   1:  PR[GP1:91,1] = PR[GP1:90,1] + -41.050;
   1:  PR[GP1:91,2] = PR[GP1:90,2] + 5.137;
   1:L PR[91] R[100]mm/sec CNT100;
   1:  PR[GP1:91,1] = PR[GP1:90,1] + -41.412;
   1:  PR[GP1:91,2] = PR[GP1:90,2] + 3.695;
   1:L PR[91] R[100]mm/sec CNT100;
   1:  PR[GP1:91,1] = PR[GP1:90,1] + -41.545;
   1:  PR[GP1:91,2] = PR[GP1:90,2] + 2.074;
   1:L PR[91] R[100]mm/sec CNT100;
   1:  PR[GP1:91,1] = PR[GP1:90,1] + -41.859;
   1:  PR[GP1:91,2] = PR[GP1:90,2] + -0.346;
   1:L PR[91] R[100]mm/sec CNT100;
   1:  PR[GP1:91,1] = PR[GP1:90,1] + -41.730;
   1:  PR[GP1:91,2] = PR[GP1:90,2] + -1.916;
   1:L PR[91] R[100]mm/sec CNT100;
   1:  PR[GP1:91,1] = PR[GP1:90,1] + -41.420;
   1:  PR[GP1:91,2] = PR[GP1:90,2] + -4.285;
   1:L PR[91] R[100]mm/sec CNT100;
   1:  PR[GP1:91,1] = PR[GP1:90,1] + -41.054;
   1:  PR[GP1:91,2] = PR[GP1:90,2] + -5.749;
   1:L PR[91] R[100]mm/sec CNT100;
   1:  PR[GP1:91,1] = PR[GP1:90,1] + -40.415;
   1:  PR[GP1:91,2] = PR[GP1:90,2] + -7.221;
   1:L PR[91] R[100]mm/sec CNT100;
   1:  PR[GP1:91,1] = PR[GP1:90,1] + -39.483;
   1:  PR[GP1:91,2] = PR[GP1:90,2] + -9.478;
   1:L PR[91] R[100]mm/sec CNT100;
   1:  PR[GP1:91,1] = PR[GP1:90,1] + -38.675;
   1:  PR[GP1:91,2] = PR[GP1:90,2] + -10.730;
   1:L PR[91] R[100]mm/sec CNT100;
   1:  PR[GP1:91,1] = PR[GP1:90,1] + -37.137;
   1:  PR[GP1:91,2] = PR[GP1:90,2] + -12.747;
   1:L PR[91] R[100]mm/sec CNT100;
   1:  PR[GP1:91,1] = PR[GP1:90,1] + -36.167;
   1:  PR[GP1:91,2] = PR[GP1:90,2] + -13.817;
   1:L PR[91] R[100]mm/sec CNT100;
   1:  PR[GP1:91,1] = PR[GP1:90,1] + -34.995;
   1:  PR[GP1:91,2] = PR[GP1:90,2] + -14.746;
   1:L PR[91] R[100]mm/sec CNT100;
   1:  PR[GP1:91,1] = PR[GP1:90,1] + -32.930;
   1:  PR[GP1:91,2] = PR[GP1:90,2] + -16.344;
   1:L PR[91] R[100]mm/sec CNT100;
   1:  PR[GP1:91,1] = PR[GP1:90,1] + -31.743;
   1:  PR[GP1:91,2] = PR[GP1:90,2] + -17.003;
   1:L PR[91] R[100]mm/sec CNT100;
   1:  PR[GP1:91,1] = PR[GP1:90,1] + -29.159;
   1:  PR[GP1:91,2] = PR[GP1:90,2] + -18.091;
   1:L PR[91] R[100]mm/sec CNT100;
   1:  PR[GP1:91,1] = PR[GP1:90,1] + -27.947;
   1:  PR[GP1:91,2] = PR[GP1:90,2] + -18.524;
   1:L PR[91] R[100]mm/sec CNT100;
   1:  PR[GP1:91,1] = PR[GP1:90,1] + -26.670;
   1:  PR[GP1:91,2] = PR[GP1:90,2] + -18.756;
   1:L PR[91] R[100]mm/sec CNT100;
   1:  PR[GP1:91,1] = PR[GP1:90,1] + -23.763;
   1:  PR[GP1:91,2] = PR[GP1:90,2] + -19.163;
   1:L PR[91] R[100]mm/sec CNT100;
   1:  PR[GP1:91,1] = PR[GP1:90,1] + -22.646;
   1:  PR[GP1:91,2] = PR[GP1:90,2] + -19.180;
   1:L PR[91] R[100]mm/sec CNT100;
   1:  PR[GP1:91,1] = PR[GP1:90,1] + -21.433;
   1:  PR[GP1:91,2] = PR[GP1:90,2] + -18.999;
   1:L PR[91] R[100]mm/sec CNT100;
   1:  PR[GP1:91,1] = PR[GP1:90,1] + -18.373;
   1:  PR[GP1:91,2] = PR[GP1:90,2] + -18.633;
   1:L PR[91] R[100]mm/sec CNT100;
   1:  PR[GP1:91,1] = PR[GP1:90,1] + -17.424;
   1:  PR[GP1:91,2] = PR[GP1:90,2] + -18.327;
   1:L PR[91] R[100]mm/sec CNT100;
   1:  PR[GP1:91,1] = PR[GP1:90,1] + -14.274;
   1:  PR[GP1:91,2] = PR[GP1:90,2] + -17.068;
   1:L PR[91] R[100]mm/sec CNT100;
   1:  PR[GP1:91,1] = PR[GP1:90,1] + -13.518;
   1:  PR[GP1:91,2] = PR[GP1:90,2] + -16.679;
   1:L PR[91] R[100]mm/sec CNT100;
   1:  PR[GP1:91,1] = PR[GP1:90,1] + -9.919;
   1:  PR[GP1:91,2] = PR[GP1:90,2] + -14.005;
   1:L PR[91] R[100]mm/sec CNT100;
   1:  PR[GP1:91,1] = PR[GP1:90,1] + -9.431;
   1:  PR[GP1:91,2] = PR[GP1:90,2] + -13.499;
   1:L PR[91] R[100]mm/sec CNT100;
   1:  PR[GP1:91,1] = PR[GP1:90,1] + -7.028;
   1:  PR[GP1:91,2] = PR[GP1:90,2] + -10.470;
   1:L PR[91] R[100]mm/sec CNT100;
   1:  PR[GP1:91,1] = PR[GP1:90,1] + -6.688;
   1:  PR[GP1:91,2] = PR[GP1:90,2] + -9.977;
   1:L PR[91] R[100]mm/sec CNT100;
   1:  PR[GP1:91,1] = PR[GP1:90,1] + -6.421;
   1:  PR[GP1:91,2] = PR[GP1:90,2] + -9.412;
   1:L PR[91] R[100]mm/sec CNT100;
   1:  PR[GP1:91,1] = PR[GP1:90,1] + -4.821;
   1:  PR[GP1:91,2] = PR[GP1:90,2] + -5.735;
   1:L PR[91] R[100]mm/sec CNT100;
   1:  PR[GP1:91,1] = PR[GP1:90,1] + -4.521;
   1:  PR[GP1:91,2] = PR[GP1:90,2] + -4.703;
   1:L PR[91] R[100]mm/sec CNT100;
   1:  PR[GP1:91,1] = PR[GP1:90,1] + -4.126;
   1:  PR[GP1:91,2] = PR[GP1:90,2] + -4.264;
   1:L PR[91] R[100]mm/sec CNT100;
   1:  PR[GP1:91,1] = PR[GP1:90,1] + -3.629;
   1:  PR[GP1:91,2] = PR[GP1:90,2] + -3.586;
   1:L PR[91] R[100]mm/sec CNT100;
   1:  PR[GP1:91,1] = PR[GP1:90,1] + -2.653;
   1:  PR[GP1:91,2] = PR[GP1:90,2] + -2.949;
   1:L PR[91] R[100]mm/sec CNT100;
   1:  PR[GP1:91,1] = PR[GP1:90,1] + -1.650;
   1:  PR[GP1:91,2] = PR[GP1:90,2] + -2.748;
   1:L PR[91] R[100]mm/sec CNT100;
   1:  PR[GP1:91,1] = PR[GP1:90,1] + 1.800;
   1:L PR[91] R[100]mm/sec CNT100;
   1:  PR[GP1:91,1] = PR[GP1:90,1] + 2.807;
   1:  PR[GP1:91,2] = PR[GP1:90,2] + -2.948;
   1:L PR[91] R[100]mm/sec CNT100;
   1:  PR[GP1:91,1] = PR[GP1:90,1] + 3.784;
   1:  PR[GP1:91,2] = PR[GP1:90,2] + -3.585;
   1:L PR[91] R[100]mm/sec CNT100;
   1:  PR[GP1:91,1] = PR[GP1:90,1] + 4.289;
   1:  PR[GP1:91,2] = PR[GP1:90,2] + -4.274;
   1:L PR[91] R[100]mm/sec CNT100;
   1:  PR[GP1:91,1] = PR[GP1:90,1] + 4.700;
   1:  PR[GP1:91,2] = PR[GP1:90,2] + -4.748;
   1:L PR[91] R[100]mm/sec CNT100;
   1:  PR[GP1:91,1] = PR[GP1:90,1] + 4.937;
   1:  PR[GP1:91,2] = PR[GP1:90,2] + -5.561;
   1:L PR[91] R[100]mm/sec CNT100;
   1:  PR[GP1:91,1] = PR[GP1:90,1] + 5.121;
   1:  PR[GP1:91,2] = PR[GP1:90,2] + -5.951;
   1:L PR[91] R[100]mm/sec CNT100;
   1:  PR[GP1:91,1] = PR[GP1:90,1] + 6.858;
   1:  PR[GP1:91,2] = PR[GP1:90,2] + -9.995;
   1:L PR[91] R[100]mm/sec CNT100;
   1:  PR[GP1:91,1] = PR[GP1:90,1] + 7.184;
   1:  PR[GP1:91,2] = PR[GP1:90,2] + -10.467;
   1:L PR[91] R[100]mm/sec CNT100;
   1:  PR[GP1:91,1] = PR[GP1:90,1] + 9.586;
   1:  PR[GP1:91,2] = PR[GP1:90,2] + -13.499;
   1:L PR[91] R[100]mm/sec CNT100;
   1:  PR[GP1:91,1] = PR[GP1:90,1] + 10.074;
   1:  PR[GP1:91,2] = PR[GP1:90,2] + -14.004;
   1:L PR[91] R[100]mm/sec CNT100;
   1:  PR[GP1:91,1] = PR[GP1:90,1] + 13.674;
   1:  PR[GP1:91,2] = PR[GP1:90,2] + -16.678;
   1:L PR[91] R[100]mm/sec CNT100;
   1:  PR[GP1:91,1] = PR[GP1:90,1] + 14.429;
   1:  PR[GP1:91,2] = PR[GP1:90,2] + -17.068;
   1:L PR[91] R[100]mm/sec CNT100;
   1:  PR[GP1:91,1] = PR[GP1:90,1] + 17.579;
   1:  PR[GP1:91,2] = PR[GP1:90,2] + -18.327;
   1:L PR[91] R[100]mm/sec CNT100;
   1:  PR[GP1:91,1] = PR[GP1:90,1] + 18.548;
   1:  PR[GP1:91,2] = PR[GP1:90,2] + -18.639;
   1:L PR[91] R[100]mm/sec CNT100;
   1:  PR[GP1:91,1] = PR[GP1:90,1] + 19.584;
   1:  PR[GP1:91,2] = PR[GP1:90,2] + -18.793;
   1:L PR[91] R[100]mm/sec CNT100;
   1:  PR[GP1:91,1] = PR[GP1:90,1] + 22.782;
   1:  PR[GP1:91,2] = PR[GP1:90,2] + -19.181;
   1:L PR[91] R[100]mm/sec CNT100;
   1:  PR[GP1:91,1] = PR[GP1:90,1] + 23.889;
   1:  PR[GP1:91,2] = PR[GP1:90,2] + -19.163;
   1:L PR[91] R[100]mm/sec CNT100;
   1:  PR[GP1:91,1] = PR[GP1:90,1] + 25.103;
   1:  PR[GP1:91,2] = PR[GP1:90,2] + -18.943;
   1:L PR[91] R[100]mm/sec CNT100;
   1:  PR[GP1:91,1] = PR[GP1:90,1] + 28.130;
   1:  PR[GP1:91,2] = PR[GP1:90,2] + -18.515;
   1:L PR[91] R[100]mm/sec CNT100;
   1:  PR[GP1:91,1] = PR[GP1:90,1] + 29.315;
   1:  PR[GP1:91,2] = PR[GP1:90,2] + -18.091;
   1:L PR[91] R[100]mm/sec CNT100;
   1:  PR[GP1:91,1] = PR[GP1:90,1] + 31.900;
   1:  PR[GP1:91,2] = PR[GP1:90,2] + -17.004;
   1:L PR[91] R[100]mm/sec CNT100;
   1:  PR[GP1:91,1] = PR[GP1:90,1] + 33.079;
   1:  PR[GP1:91,2] = PR[GP1:90,2] + -16.349;
   1:L PR[91] R[100]mm/sec CNT100;
   1:  PR[GP1:91,1] = PR[GP1:90,1] + 34.204;
   1:  PR[GP1:91,2] = PR[GP1:90,2] + -15.457;
   1:L PR[91] R[100]mm/sec CNT100;
   1:  PR[GP1:91,1] = PR[GP1:90,1] + 36.329;
   1:  PR[GP1:91,2] = PR[GP1:90,2] + -13.811;
   1:L PR[91] R[100]mm/sec CNT100;
   1:  PR[GP1:91,1] = PR[GP1:90,1] + 37.293;
   1:  PR[GP1:91,2] = PR[GP1:90,2] + -12.748;
   1:L PR[91] R[100]mm/sec CNT100;
   1:  PR[GP1:91,1] = PR[GP1:90,1] + 38.832;
   1:  PR[GP1:91,2] = PR[GP1:90,2] + -10.730;
   1:L PR[91] R[100]mm/sec CNT100;
   1:  PR[GP1:91,1] = PR[GP1:90,1] + 39.647;
   1:  PR[GP1:91,2] = PR[GP1:90,2] + -9.467;
   1:L PR[91] R[100]mm/sec CNT100;
   1:  PR[GP1:91,1] = PR[GP1:90,1] + 40.262;
   1:  PR[GP1:91,2] = PR[GP1:90,2] + -8.047;
   1:L PR[91] R[100]mm/sec CNT100;
   1:  PR[GP1:91,1] = PR[GP1:90,1] + 41.207;
   1:  PR[GP1:91,2] = PR[GP1:90,2] + -5.762;
   1:L PR[91] R[100]mm/sec CNT100;
   1:  PR[GP1:91,1] = PR[GP1:90,1] + 41.569;
   1:  PR[GP1:91,2] = PR[GP1:90,2] + -4.320;
   1:L PR[91] R[100]mm/sec CNT100;
   1:  PR[GP1:91,1] = PR[GP1:90,1] + 41.702;
   1:  PR[GP1:91,2] = PR[GP1:90,2] + -2.699;
   1:L PR[91] R[100]mm/sec CNT100;
   1:  PR[GP1:91,1] = PR[GP1:90,1] + 42.016;
   1:  PR[GP1:91,2] = PR[GP1:90,2] + -0.278;
   1:L PR[91] R[100]mm/sec CNT100;
   1:  PR[GP1:91,1] = PR[GP1:90,1] + 41.887;
   1:  PR[GP1:91,2] = PR[GP1:90,2] + 1.292;
   1:L PR[91] R[100]mm/sec CNT100;
   1:  PR[GP1:91,1] = PR[GP1:90,1] + 41.577;
   1:  PR[GP1:91,2] = PR[GP1:90,2] + 3.663;
   1:L PR[91] R[100]mm/sec CNT100;
   1:  PR[GP1:91,1] = PR[GP1:90,1] + 41.210;
   1:  PR[GP1:91,2] = PR[GP1:90,2] + 5.127;
   1:L PR[91] R[100]mm/sec CNT100;
   1:  PR[GP1:91,1] = PR[GP1:90,1] + 40.572;
   1:  PR[GP1:91,2] = PR[GP1:90,2] + 6.599;
   1:L PR[91] R[100]mm/sec CNT100;
   1:  PR[GP1:91,1] = PR[GP1:90,1] + 39.639;
   1:  PR[GP1:91,2] = PR[GP1:90,2] + 8.854;
   1:L PR[91] R[100]mm/sec CNT100;
   1:  PR[GP1:91,1] = PR[GP1:90,1] + 38.831;
   1:  PR[GP1:91,2] = PR[GP1:90,2] + 10.107;
   1:L PR[91] R[100]mm/sec CNT100;
   1:  PR[GP1:91,1] = PR[GP1:90,1] + 37.292;
   1:  PR[GP1:91,2] = PR[GP1:90,2] + 12.125;
   1:L PR[91] R[100]mm/sec CNT100;
   1:  PR[GP1:91,1] = PR[GP1:90,1] + 36.322;
   1:  PR[GP1:91,2] = PR[GP1:90,2] + 13.194;
   1:L PR[91] R[100]mm/sec CNT100;
   1:  PR[GP1:91,1] = PR[GP1:90,1] + 35.150;
   1:  PR[GP1:91,2] = PR[GP1:90,2] + 14.124;
   1:L PR[91] R[100]mm/sec CNT100;
   1:  PR[GP1:91,1] = PR[GP1:90,1] + 33.085;
   1:  PR[GP1:91,2] = PR[GP1:90,2] + 15.722;
   1:L PR[91] R[100]mm/sec CNT100;
   1:  PR[GP1:91,1] = PR[GP1:90,1] + 31.898;
   1:  PR[GP1:91,2] = PR[GP1:90,2] + 16.381;
   1:L PR[91] R[100]mm/sec CNT100;
   1:  PR[GP1:91,1] = PR[GP1:90,1] + 29.312;
   1:  PR[GP1:91,2] = PR[GP1:90,2] + 17.468;
   1:L PR[91] R[100]mm/sec CNT100;
   1:  PR[GP1:91,1] = PR[GP1:90,1] + 28.100;
   1:  PR[GP1:91,2] = PR[GP1:90,2] + 17.901;
   1:L PR[91] R[100]mm/sec CNT100;
   1:  PR[GP1:91,1] = PR[GP1:90,1] + 26.823;
   1:  PR[GP1:91,2] = PR[GP1:90,2] + 18.133;
   1:L PR[91] R[100]mm/sec CNT100;
   1:  PR[GP1:91,1] = PR[GP1:90,1] + 23.914;
   1:  PR[GP1:91,2] = PR[GP1:90,2] + 18.539;
   1:L PR[91] R[100]mm/sec CNT100;
   1:  PR[GP1:91,1] = PR[GP1:90,1] + 22.798;
   1:  PR[GP1:91,2] = PR[GP1:90,2] + 18.556;
   1:L PR[91] R[100]mm/sec CNT100;
   1:  PR[GP1:91,1] = PR[GP1:90,1] + 21.585;
   1:  PR[GP1:91,2] = PR[GP1:90,2] + 18.376;
   1:L PR[91] R[100]mm/sec CNT100;
   1:  PR[GP1:91,1] = PR[GP1:90,1] + 18.523;
   1:  PR[GP1:91,2] = PR[GP1:90,2] + 18.007;
   1:L PR[91] R[100]mm/sec CNT100;
   1:  PR[GP1:91,1] = PR[GP1:90,1] + 17.575;
   1:  PR[GP1:91,2] = PR[GP1:90,2] + 17.702;
   1:L PR[91] R[100]mm/sec CNT100;
   1:  PR[GP1:91,1] = PR[GP1:90,1] + 14.424;
   1:  PR[GP1:91,2] = PR[GP1:90,2] + 16.440;
   1:L PR[91] R[100]mm/sec CNT100;
   1:  PR[GP1:91,1] = PR[GP1:90,1] + 13.668;
   1:  PR[GP1:91,2] = PR[GP1:90,2] + 16.051;
   1:L PR[91] R[100]mm/sec CNT100;
   1:  PR[GP1:91,1] = PR[GP1:90,1] + 10.069;
   1:  PR[GP1:91,2] = PR[GP1:90,2] + 13.375;
   1:L PR[91] R[100]mm/sec CNT100;
   1:  PR[GP1:91,1] = PR[GP1:90,1] + 9.581;
   1:  PR[GP1:91,2] = PR[GP1:90,2] + 12.870;
   1:L PR[91] R[100]mm/sec CNT100;
   1:  PR[GP1:91,1] = PR[GP1:90,1] + 7.180;
   1:  PR[GP1:91,2] = PR[GP1:90,2] + 9.836;
   1:L PR[91] R[100]mm/sec CNT100;
   1:  PR[GP1:91,1] = PR[GP1:90,1] + 6.839;
   1:  PR[GP1:91,2] = PR[GP1:90,2] + 9.342;
   1:L PR[91] R[100]mm/sec CNT100;
   1:  PR[GP1:91,1] = PR[GP1:90,1] + 6.571;
   1:  PR[GP1:91,2] = PR[GP1:90,2] + 8.775;
   1:L PR[91] R[100]mm/sec CNT100;
   1:  PR[GP1:91,1] = PR[GP1:90,1] + 4.996;
   1:  PR[GP1:91,2] = PR[GP1:90,2] + 5.191;
   1:L PR[91] R[100]mm/sec CNT100;
   1:  PR[GP1:91,1] = PR[GP1:90,1] + 4.809;
   1:  PR[GP1:91,2] = PR[GP1:90,2] + 4.511;
   1:L PR[91] R[100]mm/sec CNT100;
   1:  PR[GP1:91,1] = PR[GP1:90,1] + 4.656;
   1:  PR[GP1:91,2] = PR[GP1:90,2] + 4.085;
   1:L PR[91] R[100]mm/sec CNT100;
   1:  PR[GP1:91,1] = PR[GP1:90,1] + 4.314;
   1:  PR[GP1:91,2] = PR[GP1:90,2] + 3.637;
   1:L PR[91] R[100]mm/sec CNT100;
   1:  PR[GP1:91,1] = PR[GP1:90,1] + 4.223;
   1:  PR[GP1:91,2] = PR[GP1:90,2] + 3.560;
   1:L PR[91] R[100]mm/sec CNT100;
   1:  PR[GP1:91,1] = PR[GP1:90,1] + 3.785;
   1:  PR[GP1:91,2] = PR[GP1:90,2] + 2.962;
   1:L PR[91] R[100]mm/sec CNT100;
   1:  PR[GP1:91,1] = PR[GP1:90,1] + 2.808;
   1:  PR[GP1:91,2] = PR[GP1:90,2] + 2.324;
   1:L PR[91] R[100]mm/sec CNT100;
   1:  PR[GP1:91,1] = PR[GP1:90,1] + 1.797;
   1:  PR[GP1:91,2] = PR[GP1:90,2] + 2.124;
   1:L PR[91] R[100]mm/sec CNT100;
   1:  PR[GP1:91,1] = PR[GP1:90,1] + -1.656;
   1:L PR[91] R[100]mm/sec CNT100;
   1:  PR[91] = PR[90];
   1:  PR[GP1:91,1] = PR[GP1:90,1] + -2.652;
   1:  PR[GP1:91,2] = PR[GP1:90,2] + 2.617;
   1:  PR[GP1:91,3] = PR[GP1:90,3] + 8.845;
   1:L PR[91] R[100]mm/sec CNT100;
   1:  PR[GP1:91,1] = PR[GP1:90,1] + -3.613;
   1:  PR[GP1:91,2] = PR[GP1:90,2] + 3.249;
   1:L PR[91] R[100]mm/sec CNT100;
   1:  PR[GP1:91,1] = PR[GP1:90,1] + -4.025;
   1:  PR[GP1:91,2] = PR[GP1:90,2] + 3.786;
   1:L PR[91] R[100]mm/sec CNT100;
   1:  PR[GP1:91,1] = PR[GP1:90,1] + -4.153;
   1:  PR[GP1:91,2] = PR[GP1:90,2] + 3.977;
   1:L PR[91] R[100]mm/sec CNT100;
   1:  PR[GP1:91,1] = PR[GP1:90,1] + -4.537;
   1:  PR[GP1:91,2] = PR[GP1:90,2] + 4.424;
   1:L PR[91] R[100]mm/sec CNT100;
   1:  PR[GP1:91,1] = PR[GP1:90,1] + -6.684;
   1:  PR[GP1:91,2] = PR[GP1:90,2] + 9.420;
   1:L PR[91] R[100]mm/sec CNT100;
   1:  PR[GP1:91,1] = PR[GP1:90,1] + -6.741;
   1:  PR[GP1:91,2] = PR[GP1:90,2] + 9.503;
   1:L PR[91] R[100]mm/sec CNT100;
   1:  PR[GP1:91,1] = PR[GP1:90,1] + -9.602;
   1:  PR[GP1:91,2] = PR[GP1:90,2] + 13.111;
   1:L PR[91] R[100]mm/sec CNT100;
   1:  PR[GP1:91,1] = PR[GP1:90,1] + -9.778;
   1:  PR[GP1:91,2] = PR[GP1:90,2] + 13.293;
   1:L PR[91] R[100]mm/sec CNT100;
   1:  PR[GP1:91,1] = PR[GP1:90,1] + -13.585;
   1:  PR[GP1:91,2] = PR[GP1:90,2] + 16.122;
   1:L PR[91] R[100]mm/sec CNT100;
   1:  PR[GP1:91,1] = PR[GP1:90,1] + -13.965;
   1:  PR[GP1:91,2] = PR[GP1:90,2] + 16.317;
   1:L PR[91] R[100]mm/sec CNT100;
   1:  PR[GP1:91,1] = PR[GP1:90,1] + -17.719;
   1:  PR[GP1:91,2] = PR[GP1:90,2] + 17.819;
   1:L PR[91] R[100]mm/sec CNT100;
   1:  PR[GP1:91,1] = PR[GP1:90,1] + -18.311;
   1:  PR[GP1:91,2] = PR[GP1:90,2] + 18.009;
   1:L PR[91] R[100]mm/sec CNT100;
   1:  PR[GP1:91,1] = PR[GP1:90,1] + -18.956;
   1:  PR[GP1:91,2] = PR[GP1:90,2] + 18.105;
   1:L PR[91] R[100]mm/sec CNT100;
   1:  PR[GP1:91,1] = PR[GP1:90,1] + -22.768;
   1:  PR[GP1:91,2] = PR[GP1:90,2] + 18.567;
   1:L PR[91] R[100]mm/sec CNT100;
   1:  PR[GP1:91,1] = PR[GP1:90,1] + -23.506;
   1:  PR[GP1:91,2] = PR[GP1:90,2] + 18.555;
   1:L PR[91] R[100]mm/sec CNT100;
   1:  PR[GP1:91,1] = PR[GP1:90,1] + -24.356;
   1:  PR[GP1:91,2] = PR[GP1:90,2] + 18.401;
   1:L PR[91] R[100]mm/sec CNT100;
   1:  PR[GP1:91,1] = PR[GP1:90,1] + -27.965;
   1:  PR[GP1:91,2] = PR[GP1:90,2] + 17.890;
   1:L PR[91] R[100]mm/sec CNT100;
   1:  PR[GP1:91,1] = PR[GP1:90,1] + -28.823;
   1:  PR[GP1:91,2] = PR[GP1:90,2] + 17.584;
   1:L PR[91] R[100]mm/sec CNT100;
   1:  PR[GP1:91,1] = PR[GP1:90,1] + -31.907;
   1:  PR[GP1:91,2] = PR[GP1:90,2] + 16.285;
   1:L PR[91] R[100]mm/sec CNT100;
   1:  PR[GP1:91,1] = PR[GP1:90,1] + -32.799;
   1:  PR[GP1:91,2] = PR[GP1:90,2] + 15.790;
   1:L PR[91] R[100]mm/sec CNT100;
   1:  PR[GP1:91,1] = PR[GP1:90,1] + -33.666;
   1:  PR[GP1:91,2] = PR[GP1:90,2] + 15.102;
   1:L PR[91] R[100]mm/sec CNT100;
   1:  PR[GP1:91,1] = PR[GP1:90,1] + -36.202;
   1:  PR[GP1:91,2] = PR[GP1:90,2] + 13.138;
   1:L PR[91] R[100]mm/sec CNT100;
   1:  PR[GP1:91,1] = PR[GP1:90,1] + -36.955;
   1:  PR[GP1:91,2] = PR[GP1:90,2] + 12.308;
   1:L PR[91] R[100]mm/sec CNT100;
   1:  PR[GP1:91,1] = PR[GP1:90,1] + -38.792;
   1:  PR[GP1:91,2] = PR[GP1:90,2] + 9.900;
   1:L PR[91] R[100]mm/sec CNT100;
   1:  PR[GP1:91,1] = PR[GP1:90,1] + -39.442;
   1:  PR[GP1:91,2] = PR[GP1:90,2] + 8.892;
   1:L PR[91] R[100]mm/sec CNT100;
   1:  PR[GP1:91,1] = PR[GP1:90,1] + -39.936;
   1:  PR[GP1:91,2] = PR[GP1:90,2] + 7.752;
   1:L PR[91] R[100]mm/sec CNT100;
   1:  PR[GP1:91,1] = PR[GP1:90,1] + -41.065;
   1:  PR[GP1:91,2] = PR[GP1:90,2] + 5.021;
   1:L PR[91] R[100]mm/sec CNT100;
   1:  PR[GP1:91,1] = PR[GP1:90,1] + -41.354;
   1:  PR[GP1:91,2] = PR[GP1:90,2] + 3.868;
   1:L PR[91] R[100]mm/sec CNT100;
   1:  PR[GP1:91,1] = PR[GP1:90,1] + -41.463;
   1:  PR[GP1:91,2] = PR[GP1:90,2] + 2.544;
   1:L PR[91] R[100]mm/sec CNT100;
   1:  PR[GP1:91,1] = PR[GP1:90,1] + -41.837;
   1:  PR[GP1:91,2] = PR[GP1:90,2] + -0.346;
   1:L PR[91] R[100]mm/sec CNT100;
   1:  PR[GP1:91,1] = PR[GP1:90,1] + -41.732;
   1:  PR[GP1:91,2] = PR[GP1:90,2] + -1.628;
   1:L PR[91] R[100]mm/sec CNT100;
   1:  PR[GP1:91,1] = PR[GP1:90,1] + -41.362;
   1:  PR[GP1:91,2] = PR[GP1:90,2] + -4.458;
   1:L PR[91] R[100]mm/sec CNT100;
   1:  PR[GP1:91,1] = PR[GP1:90,1] + -41.068;
   1:  PR[GP1:91,2] = PR[GP1:90,2] + -5.633;
   1:L PR[91] R[100]mm/sec CNT100;
   1:  PR[GP1:91,1] = PR[GP1:90,1] + -40.548;
   1:  PR[GP1:91,2] = PR[GP1:90,2] + -6.832;
   1:L PR[91] R[100]mm/sec CNT100;
   1:  PR[GP1:91,1] = PR[GP1:90,1] + -39.435;
   1:  PR[GP1:91,2] = PR[GP1:90,2] + -9.527;
   1:L PR[91] R[100]mm/sec CNT100;
   1:  PR[GP1:91,1] = PR[GP1:90,1] + -38.792;
   1:  PR[GP1:91,2] = PR[GP1:90,2] + -10.524;
   1:L PR[91] R[100]mm/sec CNT100;
   1:  PR[GP1:91,1] = PR[GP1:90,1] + -36.955;
   1:  PR[GP1:91,2] = PR[GP1:90,2] + -12.932;
   1:L PR[91] R[100]mm/sec CNT100;
   1:  PR[GP1:91,1] = PR[GP1:90,1] + -36.197;
   1:  PR[GP1:91,2] = PR[GP1:90,2] + -13.768;
   1:L PR[91] R[100]mm/sec CNT100;
   1:  PR[GP1:91,1] = PR[GP1:90,1] + -35.271;
   1:  PR[GP1:91,2] = PR[GP1:90,2] + -14.502;
   1:L PR[91] R[100]mm/sec CNT100;
   1:  PR[GP1:91,1] = PR[GP1:90,1] + -32.806;
   1:  PR[GP1:91,2] = PR[GP1:90,2] + -16.410;
   1:L PR[91] R[100]mm/sec CNT100;
   1:  PR[GP1:91,1] = PR[GP1:90,1] + -31.907;
   1:  PR[GP1:91,2] = PR[GP1:90,2] + -16.909;
   1:L PR[91] R[100]mm/sec CNT100;
   1:  PR[GP1:91,1] = PR[GP1:90,1] + -28.824;
   1:  PR[GP1:91,2] = PR[GP1:90,2] + -18.208;
   1:L PR[91] R[100]mm/sec CNT100;
   1:  PR[GP1:91,1] = PR[GP1:90,1] + -27.939;
   1:  PR[GP1:91,2] = PR[GP1:90,2] + -18.524;
   1:L PR[91] R[100]mm/sec CNT100;
   1:  PR[GP1:91,1] = PR[GP1:90,1] + -27.003;
   1:  PR[GP1:91,2] = PR[GP1:90,2] + -18.694;
   1:L PR[91] R[100]mm/sec CNT100;
   1:  PR[GP1:91,1] = PR[GP1:90,1] + -23.536;
   1:  PR[GP1:91,2] = PR[GP1:90,2] + -19.179;
   1:L PR[91] R[100]mm/sec CNT100;
   1:  PR[GP1:91,1] = PR[GP1:90,1] + -22.789;
   1:  PR[GP1:91,2] = PR[GP1:90,2] + -19.190;
   1:L PR[91] R[100]mm/sec CNT100;
   1:  PR[GP1:91,1] = PR[GP1:90,1] + -21.941;
   1:  PR[GP1:91,2] = PR[GP1:90,2] + -19.064;
   1:L PR[91] R[100]mm/sec CNT100;
   1:  PR[GP1:91,1] = PR[GP1:90,1] + -18.292;
   1:  PR[GP1:91,2] = PR[GP1:90,2] + -18.627;
   1:L PR[91] R[100]mm/sec CNT100;
   1:  PR[GP1:91,1] = PR[GP1:90,1] + -17.720;
   1:  PR[GP1:91,2] = PR[GP1:90,2] + -18.443;
   1:L PR[91] R[100]mm/sec CNT100;
   1:  PR[GP1:91,1] = PR[GP1:90,1] + -13.966;
   1:  PR[GP1:91,2] = PR[GP1:90,2] + -16.942;
   1:L PR[91] R[100]mm/sec CNT100;
   1:  PR[GP1:91,1] = PR[GP1:90,1] + -13.586;
   1:  PR[GP1:91,2] = PR[GP1:90,2] + -16.746;
   1:L PR[91] R[100]mm/sec CNT100;
   1:  PR[GP1:91,1] = PR[GP1:90,1] + -9.778;
   1:  PR[GP1:91,2] = PR[GP1:90,2] + -13.917;
   1:L PR[91] R[100]mm/sec CNT100;
   1:  PR[GP1:91,1] = PR[GP1:90,1] + -9.603;
   1:  PR[GP1:91,2] = PR[GP1:90,2] + -13.736;
   1:L PR[91] R[100]mm/sec CNT100;
   1:  PR[GP1:91,1] = PR[GP1:90,1] + -6.742;
   1:  PR[GP1:91,2] = PR[GP1:90,2] + -10.128;
   1:L PR[91] R[100]mm/sec CNT100;
   1:  PR[GP1:91,1] = PR[GP1:90,1] + -6.682;
   1:  PR[GP1:91,2] = PR[GP1:90,2] + -10.041;
   1:L PR[91] R[100]mm/sec CNT100;
   1:  PR[GP1:91,1] = PR[GP1:90,1] + -4.700;
   1:  PR[GP1:91,2] = PR[GP1:90,2] + -5.509;
   1:L PR[91] R[100]mm/sec CNT100;
   1:  PR[GP1:91,1] = PR[GP1:90,1] + -4.569;
   1:  PR[GP1:91,2] = PR[GP1:90,2] + -5.060;
   1:L PR[91] R[100]mm/sec CNT100;
   1:  PR[GP1:91,1] = PR[GP1:90,1] + -4.143;
   1:  PR[GP1:91,2] = PR[GP1:90,2] + -4.587;
   1:L PR[91] R[100]mm/sec CNT100;
   1:  PR[GP1:91,1] = PR[GP1:90,1] + -4.025;
   1:  PR[GP1:91,2] = PR[GP1:90,2] + -4.410;
   1:L PR[91] R[100]mm/sec CNT100;
   1:  PR[GP1:91,1] = PR[GP1:90,1] + -3.613;
   1:  PR[GP1:91,2] = PR[GP1:90,2] + -3.873;
   1:L PR[91] R[100]mm/sec CNT100;
   1:  PR[GP1:91,1] = PR[GP1:90,1] + -2.650;
   1:  PR[GP1:91,2] = PR[GP1:90,2] + -3.240;
   1:L PR[91] R[100]mm/sec CNT100;
   1:  PR[GP1:91,1] = PR[GP1:90,1] + -1.644;
   1:  PR[GP1:91,2] = PR[GP1:90,2] + -3.036;
   1:L PR[91] R[100]mm/sec CNT100;
   1:  PR[GP1:91,1] = PR[GP1:90,1] + 1.793;
   1:L PR[91] R[100]mm/sec CNT100;
   1:  PR[GP1:91,1] = PR[GP1:90,1] + 2.805;
   1:  PR[GP1:91,2] = PR[GP1:90,2] + -3.239;
   1:L PR[91] R[100]mm/sec CNT100;
   1:  PR[GP1:91,1] = PR[GP1:90,1] + 3.768;
   1:  PR[GP1:91,2] = PR[GP1:90,2] + -3.872;
   1:L PR[91] R[100]mm/sec CNT100;
   1:  PR[GP1:91,1] = PR[GP1:90,1] + 4.180;
   1:  PR[GP1:91,2] = PR[GP1:90,2] + -4.409;
   1:L PR[91] R[100]mm/sec CNT100;
   1:  PR[GP1:91,1] = PR[GP1:90,1] + 4.305;
   1:  PR[GP1:91,2] = PR[GP1:90,2] + -4.597;
   1:L PR[91] R[100]mm/sec CNT100;
   1:  PR[GP1:91,1] = PR[GP1:90,1] + 4.694;
   1:  PR[GP1:91,2] = PR[GP1:90,2] + -5.045;
   1:L PR[91] R[100]mm/sec CNT100;
   1:  PR[GP1:91,1] = PR[GP1:90,1] + 6.840;
   1:  PR[GP1:91,2] = PR[GP1:90,2] + -10.042;
   1:L PR[91] R[100]mm/sec CNT100;
   1:  PR[GP1:91,1] = PR[GP1:90,1] + 6.897;
   1:  PR[GP1:91,2] = PR[GP1:90,2] + -10.124;
   1:L PR[91] R[100]mm/sec CNT100;
   1:  PR[GP1:91,1] = PR[GP1:90,1] + 9.758;
   1:  PR[GP1:91,2] = PR[GP1:90,2] + -13.735;
   1:L PR[91] R[100]mm/sec CNT100;
   1:  PR[GP1:91,1] = PR[GP1:90,1] + 9.934;
   1:  PR[GP1:91,2] = PR[GP1:90,2] + -13.916;
   1:L PR[91] R[100]mm/sec CNT100;
   1:  PR[GP1:91,1] = PR[GP1:90,1] + 13.741;
   1:  PR[GP1:91,2] = PR[GP1:90,2] + -16.746;
   1:L PR[91] R[100]mm/sec CNT100;
   1:  PR[GP1:91,1] = PR[GP1:90,1] + 14.121;
   1:  PR[GP1:91,2] = PR[GP1:90,2] + -16.941;
   1:L PR[91] R[100]mm/sec CNT100;
   1:  PR[GP1:91,1] = PR[GP1:90,1] + 17.875;
   1:  PR[GP1:91,2] = PR[GP1:90,2] + -18.442;
   1:L PR[91] R[100]mm/sec CNT100;
   1:  PR[GP1:91,1] = PR[GP1:90,1] + 18.467;
   1:  PR[GP1:91,2] = PR[GP1:90,2] + -18.633;
   1:L PR[91] R[100]mm/sec CNT100;
   1:  PR[GP1:91,1] = PR[GP1:90,1] + 19.112;
   1:  PR[GP1:91,2] = PR[GP1:90,2] + -18.729;
   1:L PR[91] R[100]mm/sec CNT100;
   1:  PR[GP1:91,1] = PR[GP1:90,1] + 22.924;
   1:  PR[GP1:91,2] = PR[GP1:90,2] + -19.191;
   1:L PR[91] R[100]mm/sec CNT100;
   1:  PR[GP1:91,1] = PR[GP1:90,1] + 23.662;
   1:  PR[GP1:91,2] = PR[GP1:90,2] + -19.179;
   1:L PR[91] R[100]mm/sec CNT100;
   1:  PR[GP1:91,1] = PR[GP1:90,1] + 24.512;
   1:  PR[GP1:91,2] = PR[GP1:90,2] + -19.025;
   1:L PR[91] R[100]mm/sec CNT100;
   1:  PR[GP1:91,1] = PR[GP1:90,1] + 28.121;
   1:  PR[GP1:91,2] = PR[GP1:90,2] + -18.514;
   1:L PR[91] R[100]mm/sec CNT100;
   1:  PR[GP1:91,1] = PR[GP1:90,1] + 28.980;
   1:  PR[GP1:91,2] = PR[GP1:90,2] + -18.208;
   1:L PR[91] R[100]mm/sec CNT100;
   1:  PR[GP1:91,1] = PR[GP1:90,1] + 32.063;
   1:  PR[GP1:91,2] = PR[GP1:90,2] + -16.910;
   1:L PR[91] R[100]mm/sec CNT100;
   1:  PR[GP1:91,1] = PR[GP1:90,1] + 32.955;
   1:  PR[GP1:91,2] = PR[GP1:90,2] + -16.415;
   1:L PR[91] R[100]mm/sec CNT100;
   1:  PR[GP1:91,1] = PR[GP1:90,1] + 33.822;
   1:  PR[GP1:91,2] = PR[GP1:90,2] + -15.727;
   1:L PR[91] R[100]mm/sec CNT100;
   1:  PR[GP1:91,1] = PR[GP1:90,1] + 36.359;
   1:  PR[GP1:91,2] = PR[GP1:90,2] + -13.763;
   1:L PR[91] R[100]mm/sec CNT100;
   1:  PR[GP1:91,1] = PR[GP1:90,1] + 37.112;
   1:  PR[GP1:91,2] = PR[GP1:90,2] + -12.932;
   1:L PR[91] R[100]mm/sec CNT100;
   1:  PR[GP1:91,1] = PR[GP1:90,1] + 38.949;
   1:  PR[GP1:91,2] = PR[GP1:90,2] + -10.523;
   1:L PR[91] R[100]mm/sec CNT100;
   1:  PR[GP1:91,1] = PR[GP1:90,1] + 39.599;
   1:  PR[GP1:91,2] = PR[GP1:90,2] + -9.515;
   1:L PR[91] R[100]mm/sec CNT100;
   1:  PR[GP1:91,1] = PR[GP1:90,1] + 40.093;
   1:  PR[GP1:91,2] = PR[GP1:90,2] + -8.375;
   1:L PR[91] R[100]mm/sec CNT100;
   1:  PR[GP1:91,1] = PR[GP1:90,1] + 41.222;
   1:  PR[GP1:91,2] = PR[GP1:90,2] + -5.647;
   1:L PR[91] R[100]mm/sec CNT100;
   1:  PR[GP1:91,1] = PR[GP1:90,1] + 41.511;
   1:  PR[GP1:91,2] = PR[GP1:90,2] + -4.494;
   1:L PR[91] R[100]mm/sec CNT100;
   1:  PR[GP1:91,1] = PR[GP1:90,1] + 41.619;
   1:  PR[GP1:91,2] = PR[GP1:90,2] + -3.170;
   1:L PR[91] R[100]mm/sec CNT100;
   1:  PR[GP1:91,1] = PR[GP1:90,1] + 41.994;
   1:  PR[GP1:91,2] = PR[GP1:90,2] + -0.278;
   1:L PR[91] R[100]mm/sec CNT100;
   1:  PR[GP1:91,1] = PR[GP1:90,1] + 41.889;
   1:  PR[GP1:91,2] = PR[GP1:90,2] + 1.004;
   1:L PR[91] R[100]mm/sec CNT100;
   1:  PR[GP1:91,1] = PR[GP1:90,1] + 41.519;
   1:  PR[GP1:91,2] = PR[GP1:90,2] + 3.837;
   1:L PR[91] R[100]mm/sec CNT100;
   1:  PR[GP1:91,1] = PR[GP1:90,1] + 41.225;
   1:  PR[GP1:91,2] = PR[GP1:90,2] + 5.011;
   1:L PR[91] R[100]mm/sec CNT100;
   1:  PR[GP1:91,1] = PR[GP1:90,1] + 40.705;
   1:  PR[GP1:91,2] = PR[GP1:90,2] + 6.210;
   1:L PR[91] R[100]mm/sec CNT100;
   1:  PR[GP1:91,1] = PR[GP1:90,1] + 39.591;
   1:  PR[GP1:91,2] = PR[GP1:90,2] + 8.903;
   1:L PR[91] R[100]mm/sec CNT100;
   1:  PR[GP1:91,1] = PR[GP1:90,1] + 38.948;
   1:  PR[GP1:91,2] = PR[GP1:90,2] + 9.900;
   1:L PR[91] R[100]mm/sec CNT100;
   1:  PR[GP1:91,1] = PR[GP1:90,1] + 37.110;
   1:  PR[GP1:91,2] = PR[GP1:90,2] + 12.310;
   1:L PR[91] R[100]mm/sec CNT100;
   1:  PR[GP1:91,1] = PR[GP1:90,1] + 36.352;
   1:  PR[GP1:91,2] = PR[GP1:90,2] + 13.146;
   1:L PR[91] R[100]mm/sec CNT100;
   1:  PR[GP1:91,1] = PR[GP1:90,1] + 35.426;
   1:  PR[GP1:91,2] = PR[GP1:90,2] + 13.881;
   1:L PR[91] R[100]mm/sec CNT100;
   1:  PR[GP1:91,1] = PR[GP1:90,1] + 32.960;
   1:  PR[GP1:91,2] = PR[GP1:90,2] + 15.788;
   1:L PR[91] R[100]mm/sec CNT100;
   1:  PR[GP1:91,1] = PR[GP1:90,1] + 32.061;
   1:  PR[GP1:91,2] = PR[GP1:90,2] + 16.287;
   1:L PR[91] R[100]mm/sec CNT100;
   1:  PR[GP1:91,1] = PR[GP1:90,1] + 28.976;
   1:  PR[GP1:91,2] = PR[GP1:90,2] + 17.585;
   1:L PR[91] R[100]mm/sec CNT100;
   1:  PR[GP1:91,1] = PR[GP1:90,1] + 28.091;
   1:  PR[GP1:91,2] = PR[GP1:90,2] + 17.901;
   1:L PR[91] R[100]mm/sec CNT100;
   1:  PR[GP1:91,1] = PR[GP1:90,1] + 27.156;
   1:  PR[GP1:91,2] = PR[GP1:90,2] + 18.071;
   1:L PR[91] R[100]mm/sec CNT100;
   1:  PR[GP1:91,1] = PR[GP1:90,1] + 23.686;
   1:  PR[GP1:91,2] = PR[GP1:90,2] + 18.555;
   1:L PR[91] R[100]mm/sec CNT100;
   1:  PR[GP1:91,1] = PR[GP1:90,1] + 22.939;
   1:  PR[GP1:91,2] = PR[GP1:90,2] + 18.566;
   1:L PR[91] R[100]mm/sec CNT100;
   1:  PR[GP1:91,1] = PR[GP1:90,1] + 22.093;
   1:  PR[GP1:91,2] = PR[GP1:90,2] + 18.440;
   1:L PR[91] R[100]mm/sec CNT100;
   1:  PR[GP1:91,1] = PR[GP1:90,1] + 18.442;
   1:  PR[GP1:91,2] = PR[GP1:90,2] + 18.001;
   1:L PR[91] R[100]mm/sec CNT100;
   1:  PR[GP1:91,1] = PR[GP1:90,1] + 17.870;
   1:  PR[GP1:91,2] = PR[GP1:90,2] + 17.817;
   1:L PR[91] R[100]mm/sec CNT100;
   1:  PR[GP1:91,1] = PR[GP1:90,1] + 14.114;
   1:  PR[GP1:91,2] = PR[GP1:90,2] + 16.314;
   1:L PR[91] R[100]mm/sec CNT100;
   1:  PR[GP1:91,1] = PR[GP1:90,1] + 13.735;
   1:  PR[GP1:91,2] = PR[GP1:90,2] + 16.118;
   1:L PR[91] R[100]mm/sec CNT100;
   1:  PR[GP1:91,1] = PR[GP1:90,1] + 9.927;
   1:  PR[GP1:91,2] = PR[GP1:90,2] + 13.286;
   1:L PR[91] R[100]mm/sec CNT100;
   1:  PR[GP1:91,1] = PR[GP1:90,1] + 9.752;
   1:  PR[GP1:91,2] = PR[GP1:90,2] + 13.105;
   1:L PR[91] R[100]mm/sec CNT100;
   1:  PR[GP1:91,1] = PR[GP1:90,1] + 6.892;
   1:  PR[GP1:91,2] = PR[GP1:90,2] + 9.491;
   1:L PR[91] R[100]mm/sec CNT100;
   1:  PR[GP1:91,1] = PR[GP1:90,1] + 6.831;
   1:  PR[GP1:91,2] = PR[GP1:90,2] + 9.403;
   1:L PR[91] R[100]mm/sec CNT100;
   1:  PR[GP1:91,1] = PR[GP1:90,1] + 4.874;
   1:  PR[GP1:91,2] = PR[GP1:90,2] + 4.969;
   1:L PR[91] R[100]mm/sec CNT100;
   1:  PR[GP1:91,1] = PR[GP1:90,1] + 4.731;
   1:  PR[GP1:91,2] = PR[GP1:90,2] + 4.476;
   1:L PR[91] R[100]mm/sec CNT100;
   1:  PR[GP1:91,1] = PR[GP1:90,1] + 4.333;
   1:  PR[GP1:91,2] = PR[GP1:90,2] + 3.956;
   1:L PR[91] R[100]mm/sec CNT100;
   1:  PR[GP1:91,1] = PR[GP1:90,1] + 4.244;
   1:  PR[GP1:91,2] = PR[GP1:90,2] + 3.880;
   1:L PR[91] R[100]mm/sec CNT100;
   1:  PR[GP1:91,1] = PR[GP1:90,1] + 4.182;
   1:  PR[GP1:91,2] = PR[GP1:90,2] + 3.787;
   1:L PR[91] R[100]mm/sec CNT100;
   1:  PR[GP1:91,1] = PR[GP1:90,1] + 3.769;
   1:  PR[GP1:91,2] = PR[GP1:90,2] + 3.249;
   1:L PR[91] R[100]mm/sec CNT100;
   1:  PR[GP1:91,1] = PR[GP1:90,1] + 2.805;
   1:  PR[GP1:91,2] = PR[GP1:90,2] + 2.615;
   1:L PR[91] R[100]mm/sec CNT100;
   1:  PR[GP1:91,1] = PR[GP1:90,1] + 1.788;
   1:  PR[GP1:91,2] = PR[GP1:90,2] + 2.412;
   1:L PR[91] R[100]mm/sec CNT100;
   1:  PR[GP1:91,1] = PR[GP1:90,1] + -1.651;
   1:L PR[91] R[100]mm/sec CNT100;
   1:  PR[91] = PR[90];
   1:  PR[GP1:91,1] = PR[GP1:90,1] + -2.650;
   1:  PR[GP1:91,2] = PR[GP1:90,2] + 2.908;
   1:  PR[GP1:91,3] = PR[GP1:90,3] + 9.455;
   1:L PR[91] R[100]mm/sec CNT100;
   1:  PR[GP1:91,1] = PR[GP1:90,1] + -3.611;
   1:  PR[GP1:91,2] = PR[GP1:90,2] + 3.545;
   1:L PR[91] R[100]mm/sec CNT100;
   1:  PR[GP1:91,1] = PR[GP1:90,1] + -3.992;
   1:  PR[GP1:91,2] = PR[GP1:90,2] + 4.042;
   1:L PR[91] R[100]mm/sec CNT100;
   1:  PR[GP1:91,1] = PR[GP1:90,1] + -4.146;
   1:  PR[GP1:91,2] = PR[GP1:90,2] + 4.272;
   1:L PR[91] R[100]mm/sec CNT100;
   1:  PR[GP1:91,1] = PR[GP1:90,1] + -4.490;
   1:  PR[GP1:91,2] = PR[GP1:90,2] + 4.667;
   1:L PR[91] R[100]mm/sec CNT100;
   1:  PR[GP1:91,1] = PR[GP1:90,1] + -6.559;
   1:  PR[GP1:91,2] = PR[GP1:90,2] + 9.328;
   1:L PR[91] R[100]mm/sec CNT100;
   1:  PR[GP1:91,1] = PR[GP1:90,1] + -6.611;
   1:  PR[GP1:91,2] = PR[GP1:90,2] + 9.425;
   1:L PR[91] R[100]mm/sec CNT100;
   1:  PR[GP1:91,1] = PR[GP1:90,1] + -9.683;
   1:  PR[GP1:91,2] = PR[GP1:90,2] + 13.238;
   1:L PR[91] R[100]mm/sec CNT100;
   1:  PR[GP1:91,1] = PR[GP1:90,1] + -13.653;
   1:  PR[GP1:91,2] = PR[GP1:90,2] + 16.189;
   1:L PR[91] R[100]mm/sec CNT100;
   1:  PR[GP1:91,1] = PR[GP1:90,1] + -13.657;
   1:  PR[GP1:91,2] = PR[GP1:90,2] + 16.191;
   1:L PR[91] R[100]mm/sec CNT100;
   1:  PR[GP1:91,1] = PR[GP1:90,1] + -18.015;
   1:  PR[GP1:91,2] = PR[GP1:90,2] + 17.934;
   1:L PR[91] R[100]mm/sec CNT100;
   1:  PR[GP1:91,1] = PR[GP1:90,1] + -18.213;
   1:  PR[GP1:91,2] = PR[GP1:90,2] + 17.998;
   1:L PR[91] R[100]mm/sec CNT100;
   1:  PR[GP1:91,1] = PR[GP1:90,1] + -22.912;
   1:  PR[GP1:91,2] = PR[GP1:90,2] + 18.577;
   1:L PR[91] R[100]mm/sec CNT100;
   1:  PR[GP1:91,1] = PR[GP1:90,1] + -23.279;
   1:  PR[GP1:91,2] = PR[GP1:90,2] + 18.571;
   1:L PR[91] R[100]mm/sec CNT100;
   1:  PR[GP1:91,1] = PR[GP1:90,1] + -23.765;
   1:  PR[GP1:91,2] = PR[GP1:90,2] + 18.483;
   1:L PR[91] R[100]mm/sec CNT100;
   1:  PR[GP1:91,1] = PR[GP1:90,1] + -27.957;
   1:  PR[GP1:91,2] = PR[GP1:90,2] + 17.890;
   1:L PR[91] R[100]mm/sec CNT100;
   1:  PR[GP1:91,1] = PR[GP1:90,1] + -28.488;
   1:  PR[GP1:91,2] = PR[GP1:90,2] + 17.700;
   1:L PR[91] R[100]mm/sec CNT100;
   1:  PR[GP1:91,1] = PR[GP1:90,1] + -32.070;
   1:  PR[GP1:91,2] = PR[GP1:90,2] + 16.192;
   1:L PR[91] R[100]mm/sec CNT100;
   1:  PR[GP1:91,1] = PR[GP1:90,1] + -32.681;
   1:  PR[GP1:91,2] = PR[GP1:90,2] + 15.853;
   1:L PR[91] R[100]mm/sec CNT100;
   1:  PR[GP1:91,1] = PR[GP1:90,1] + -36.231;
   1:  PR[GP1:91,2] = PR[GP1:90,2] + 13.091;
   1:L PR[91] R[100]mm/sec CNT100;
   1:  PR[GP1:91,1] = PR[GP1:90,1] + -36.773;
   1:  PR[GP1:91,2] = PR[GP1:90,2] + 12.493;
   1:L PR[91] R[100]mm/sec CNT100;
   1:  PR[GP1:91,1] = PR[GP1:90,1] + -38.909;
   1:  PR[GP1:91,2] = PR[GP1:90,2] + 9.693;
   1:L PR[91] R[100]mm/sec CNT100;
   1:  PR[GP1:91,1] = PR[GP1:90,1] + -39.394;
   1:  PR[GP1:91,2] = PR[GP1:90,2] + 8.941;
   1:L PR[91] R[100]mm/sec CNT100;
   1:  PR[GP1:91,1] = PR[GP1:90,1] + -39.768;
   1:  PR[GP1:91,2] = PR[GP1:90,2] + 8.080;
   1:L PR[91] R[100]mm/sec CNT100;
   1:  PR[GP1:91,1] = PR[GP1:90,1] + -41.079;
   1:  PR[GP1:91,2] = PR[GP1:90,2] + 4.905;
   1:L PR[91] R[100]mm/sec CNT100;
   1:  PR[GP1:91,1] = PR[GP1:90,1] + -41.296;
   1:  PR[GP1:91,2] = PR[GP1:90,2] + 4.041;
   1:L PR[91] R[100]mm/sec CNT100;
   1:  PR[GP1:91,1] = PR[GP1:90,1] + -41.380;
   1:  PR[GP1:91,2] = PR[GP1:90,2] + 3.014;
   1:L PR[91] R[100]mm/sec CNT100;
   1:  PR[GP1:91,1] = PR[GP1:90,1] + -41.816;
   1:  PR[GP1:91,2] = PR[GP1:90,2] + -0.346;
   1:L PR[91] R[100]mm/sec CNT100;
   1:  PR[GP1:91,1] = PR[GP1:90,1] + -41.734;
   1:  PR[GP1:91,2] = PR[GP1:90,2] + -1.340;
   1:L PR[91] R[100]mm/sec CNT100;
   1:  PR[GP1:91,1] = PR[GP1:90,1] + -41.304;
   1:  PR[GP1:91,2] = PR[GP1:90,2] + -4.631;
   1:L PR[91] R[100]mm/sec CNT100;
   1:  PR[GP1:91,1] = PR[GP1:90,1] + -41.083;
   1:  PR[GP1:91,2] = PR[GP1:90,2] + -5.516;
   1:L PR[91] R[100]mm/sec CNT100;
   1:  PR[GP1:91,1] = PR[GP1:90,1] + -40.681;
   1:  PR[GP1:91,2] = PR[GP1:90,2] + -6.442;
   1:L PR[91] R[100]mm/sec CNT100;
   1:  PR[GP1:91,1] = PR[GP1:90,1] + -39.387;
   1:  PR[GP1:91,2] = PR[GP1:90,2] + -9.576;
   1:L PR[91] R[100]mm/sec CNT100;
   1:  PR[GP1:91,1] = PR[GP1:90,1] + -38.909;
   1:  PR[GP1:91,2] = PR[GP1:90,2] + -10.317;
   1:L PR[91] R[100]mm/sec CNT100;
   1:  PR[GP1:91,1] = PR[GP1:90,1] + -36.774;
   1:  PR[GP1:91,2] = PR[GP1:90,2] + -13.116;
   1:L PR[91] R[100]mm/sec CNT100;
   1:  PR[GP1:91,1] = PR[GP1:90,1] + -36.231;
   1:  PR[GP1:91,2] = PR[GP1:90,2] + -13.715;
   1:L PR[91] R[100]mm/sec CNT100;
   1:  PR[GP1:91,1] = PR[GP1:90,1] + -32.681;
   1:  PR[GP1:91,2] = PR[GP1:90,2] + -16.476;
   1:L PR[91] R[100]mm/sec CNT100;
   1:  PR[GP1:91,1] = PR[GP1:90,1] + -32.071;
   1:  PR[GP1:91,2] = PR[GP1:90,2] + -16.815;
   1:L PR[91] R[100]mm/sec CNT100;
   1:  PR[GP1:91,1] = PR[GP1:90,1] + -28.488;
   1:  PR[GP1:91,2] = PR[GP1:90,2] + -18.324;
   1:L PR[91] R[100]mm/sec CNT100;
   1:  PR[GP1:91,1] = PR[GP1:90,1] + -27.930;
   1:  PR[GP1:91,2] = PR[GP1:90,2] + -18.523;
   1:L PR[91] R[100]mm/sec CNT100;
   1:  PR[GP1:91,1] = PR[GP1:90,1] + -27.337;
   1:  PR[GP1:91,2] = PR[GP1:90,2] + -18.631;
   1:L PR[91] R[100]mm/sec CNT100;
   1:  PR[GP1:91,1] = PR[GP1:90,1] + -23.308;
   1:  PR[GP1:91,2] = PR[GP1:90,2] + -19.194;
   1:L PR[91] R[100]mm/sec CNT100;
   1:  PR[GP1:91,1] = PR[GP1:90,1] + -22.931;
   1:  PR[GP1:91,2] = PR[GP1:90,2] + -19.200;
   1:L PR[91] R[100]mm/sec CNT100;
   1:  PR[GP1:91,1] = PR[GP1:90,1] + -22.450;
   1:  PR[GP1:91,2] = PR[GP1:90,2] + -19.129;
   1:L PR[91] R[100]mm/sec CNT100;
   1:  PR[GP1:91,1] = PR[GP1:90,1] + -18.211;
   1:  PR[GP1:91,2] = PR[GP1:90,2] + -18.621;
   1:L PR[91] R[100]mm/sec CNT100;
   1:  PR[GP1:91,1] = PR[GP1:90,1] + -18.016;
   1:  PR[GP1:91,2] = PR[GP1:90,2] + -18.558;
   1:L PR[91] R[100]mm/sec CNT100;
   1:  PR[GP1:91,1] = PR[GP1:90,1] + -13.658;
   1:  PR[GP1:91,2] = PR[GP1:90,2] + -16.816;
   1:L PR[91] R[100]mm/sec CNT100;
   1:  PR[GP1:91,1] = PR[GP1:90,1] + -13.654;
   1:  PR[GP1:91,2] = PR[GP1:90,2] + -16.814;
   1:L PR[91] R[100]mm/sec CNT100;
   1:  PR[GP1:91,1] = PR[GP1:90,1] + -9.694;
   1:  PR[GP1:91,2] = PR[GP1:90,2] + -13.873;
   1:L PR[91] R[100]mm/sec CNT100;
   1:  PR[GP1:91,1] = PR[GP1:90,1] + -6.612;
   1:  PR[GP1:91,2] = PR[GP1:90,2] + -10.049;
   1:L PR[91] R[100]mm/sec CNT100;
   1:  PR[GP1:91,1] = PR[GP1:90,1] + -6.560;
   1:  PR[GP1:91,2] = PR[GP1:90,2] + -9.954;
   1:L PR[91] R[100]mm/sec CNT100;
   1:  PR[GP1:91,1] = PR[GP1:90,1] + -4.495;
   1:  PR[GP1:91,2] = PR[GP1:90,2] + -5.278;
   1:L PR[91] R[100]mm/sec CNT100;
   1:  PR[GP1:91,1] = PR[GP1:90,1] + -4.138;
   1:  PR[GP1:91,2] = PR[GP1:90,2] + -4.884;
   1:L PR[91] R[100]mm/sec CNT100;
   1:  PR[GP1:91,1] = PR[GP1:90,1] + -3.992;
   1:  PR[GP1:91,2] = PR[GP1:90,2] + -4.666;
   1:L PR[91] R[100]mm/sec CNT100;
   1:  PR[GP1:91,1] = PR[GP1:90,1] + -3.611;
   1:  PR[GP1:91,2] = PR[GP1:90,2] + -4.168;
   1:L PR[91] R[100]mm/sec CNT100;
   1:  PR[GP1:91,1] = PR[GP1:90,1] + -2.648;
   1:  PR[GP1:91,2] = PR[GP1:90,2] + -3.531;
   1:L PR[91] R[100]mm/sec CNT100;
   1:  PR[GP1:91,1] = PR[GP1:90,1] + -1.638;
   1:  PR[GP1:91,2] = PR[GP1:90,2] + -3.325;
   1:L PR[91] R[100]mm/sec CNT100;
   1:  PR[GP1:91,1] = PR[GP1:90,1] + 1.785;
   1:L PR[91] R[100]mm/sec CNT100;
   1:  PR[GP1:91,1] = PR[GP1:90,1] + 2.802;
   1:  PR[GP1:91,2] = PR[GP1:90,2] + -3.530;
   1:L PR[91] R[100]mm/sec CNT100;
   1:  PR[GP1:91,1] = PR[GP1:90,1] + 3.765;
   1:  PR[GP1:91,2] = PR[GP1:90,2] + -4.167;
   1:L PR[91] R[100]mm/sec CNT100;
   1:  PR[GP1:91,1] = PR[GP1:90,1] + 4.147;
   1:  PR[GP1:91,2] = PR[GP1:90,2] + -4.665;
   1:L PR[91] R[100]mm/sec CNT100;
   1:  PR[GP1:91,1] = PR[GP1:90,1] + 4.299;
   1:  PR[GP1:91,2] = PR[GP1:90,2] + -4.893;
   1:L PR[91] R[100]mm/sec CNT100;
   1:  PR[GP1:91,1] = PR[GP1:90,1] + 4.646;
   1:  PR[GP1:91,2] = PR[GP1:90,2] + -5.289;
   1:L PR[91] R[100]mm/sec CNT100;
   1:  PR[GP1:91,1] = PR[GP1:90,1] + 6.714;
   1:  PR[GP1:91,2] = PR[GP1:90,2] + -9.948;
   1:L PR[91] R[100]mm/sec CNT100;
   1:  PR[GP1:91,1] = PR[GP1:90,1] + 6.767;
   1:  PR[GP1:91,2] = PR[GP1:90,2] + -10.045;
   1:L PR[91] R[100]mm/sec CNT100;
   1:  PR[GP1:91,1] = PR[GP1:90,1] + 9.839;
   1:  PR[GP1:91,2] = PR[GP1:90,2] + -13.861;
   1:L PR[91] R[100]mm/sec CNT100;
   1:  PR[GP1:91,1] = PR[GP1:90,1] + 13.809;
   1:  PR[GP1:91,2] = PR[GP1:90,2] + -16.813;
   1:L PR[91] R[100]mm/sec CNT100;
   1:  PR[GP1:91,1] = PR[GP1:90,1] + 13.813;
   1:  PR[GP1:91,2] = PR[GP1:90,2] + -16.815;
   1:L PR[91] R[100]mm/sec CNT100;
   1:  PR[GP1:91,1] = PR[GP1:90,1] + 18.171;
   1:  PR[GP1:91,2] = PR[GP1:90,2] + -18.557;
   1:L PR[91] R[100]mm/sec CNT100;
   1:  PR[GP1:91,1] = PR[GP1:90,1] + 18.387;
   1:  PR[GP1:91,2] = PR[GP1:90,2] + -18.627;
   1:L PR[91] R[100]mm/sec CNT100;
   1:  PR[GP1:91,1] = PR[GP1:90,1] + 18.640;
   1:  PR[GP1:91,2] = PR[GP1:90,2] + -18.665;
   1:L PR[91] R[100]mm/sec CNT100;
   1:  PR[GP1:91,1] = PR[GP1:90,1] + 23.067;
   1:  PR[GP1:91,2] = PR[GP1:90,2] + -19.201;
   1:L PR[91] R[100]mm/sec CNT100;
   1:  PR[GP1:91,1] = PR[GP1:90,1] + 23.435;
   1:  PR[GP1:91,2] = PR[GP1:90,2] + -19.195;
   1:L PR[91] R[100]mm/sec CNT100;
   1:  PR[GP1:91,1] = PR[GP1:90,1] + 23.921;
   1:  PR[GP1:91,2] = PR[GP1:90,2] + -19.107;
   1:L PR[91] R[100]mm/sec CNT100;
   1:  PR[GP1:91,1] = PR[GP1:90,1] + 28.113;
   1:  PR[GP1:91,2] = PR[GP1:90,2] + -18.514;
   1:L PR[91] R[100]mm/sec CNT100;
   1:  PR[GP1:91,1] = PR[GP1:90,1] + 28.644;
   1:  PR[GP1:91,2] = PR[GP1:90,2] + -18.324;
   1:L PR[91] R[100]mm/sec CNT100;
   1:  PR[GP1:91,1] = PR[GP1:90,1] + 32.227;
   1:  PR[GP1:91,2] = PR[GP1:90,2] + -16.816;
   1:L PR[91] R[100]mm/sec CNT100;
   1:  PR[GP1:91,1] = PR[GP1:90,1] + 32.837;
   1:  PR[GP1:91,2] = PR[GP1:90,2] + -16.477;
   1:L PR[91] R[100]mm/sec CNT100;
   1:  PR[GP1:91,1] = PR[GP1:90,1] + 36.387;
   1:  PR[GP1:91,2] = PR[GP1:90,2] + -13.715;
   1:L PR[91] R[100]mm/sec CNT100;
   1:  PR[GP1:91,1] = PR[GP1:90,1] + 36.930;
   1:  PR[GP1:91,2] = PR[GP1:90,2] + -13.117;
   1:L PR[91] R[100]mm/sec CNT100;
   1:  PR[GP1:91,1] = PR[GP1:90,1] + 39.066;
   1:  PR[GP1:91,2] = PR[GP1:90,2] + -10.316;
   1:L PR[91] R[100]mm/sec CNT100;
   1:  PR[GP1:91,1] = PR[GP1:90,1] + 39.551;
   1:  PR[GP1:91,2] = PR[GP1:90,2] + -9.564;
   1:L PR[91] R[100]mm/sec CNT100;
   1:  PR[GP1:91,1] = PR[GP1:90,1] + 39.924;
   1:  PR[GP1:91,2] = PR[GP1:90,2] + -8.703;
   1:L PR[91] R[100]mm/sec CNT100;
   1:  PR[GP1:91,1] = PR[GP1:90,1] + 41.236;
   1:  PR[GP1:91,2] = PR[GP1:90,2] + -5.531;
   1:L PR[91] R[100]mm/sec CNT100;
   1:  PR[GP1:91,1] = PR[GP1:90,1] + 41.453;
   1:  PR[GP1:91,2] = PR[GP1:90,2] + -4.667;
   1:L PR[91] R[100]mm/sec CNT100;
   1:  PR[GP1:91,1] = PR[GP1:90,1] + 41.537;
   1:  PR[GP1:91,2] = PR[GP1:90,2] + -3.641;
   1:L PR[91] R[100]mm/sec CNT100;
   1:  PR[GP1:91,1] = PR[GP1:90,1] + 41.973;
   1:  PR[GP1:91,2] = PR[GP1:90,2] + -0.278;
   1:L PR[91] R[100]mm/sec CNT100;
   1:  PR[GP1:91,1] = PR[GP1:90,1] + 41.891;
   1:  PR[GP1:91,2] = PR[GP1:90,2] + 0.716;
   1:L PR[91] R[100]mm/sec CNT100;
   1:  PR[GP1:91,1] = PR[GP1:90,1] + 41.461;
   1:  PR[GP1:91,2] = PR[GP1:90,2] + 4.010;
   1:L PR[91] R[100]mm/sec CNT100;
   1:  PR[GP1:91,1] = PR[GP1:90,1] + 41.239;
   1:  PR[GP1:91,2] = PR[GP1:90,2] + 4.896;
   1:L PR[91] R[100]mm/sec CNT100;
   1:  PR[GP1:91,1] = PR[GP1:90,1] + 40.838;
   1:  PR[GP1:91,2] = PR[GP1:90,2] + 5.821;
   1:L PR[91] R[100]mm/sec CNT100;
   1:  PR[GP1:91,1] = PR[GP1:90,1] + 39.543;
   1:  PR[GP1:91,2] = PR[GP1:90,2] + 8.952;
   1:L PR[91] R[100]mm/sec CNT100;
   1:  PR[GP1:91,1] = PR[GP1:90,1] + 39.065;
   1:  PR[GP1:91,2] = PR[GP1:90,2] + 9.693;
   1:L PR[91] R[100]mm/sec CNT100;
   1:  PR[GP1:91,1] = PR[GP1:90,1] + 36.928;
   1:  PR[GP1:91,2] = PR[GP1:90,2] + 12.495;
   1:L PR[91] R[100]mm/sec CNT100;
   1:  PR[GP1:91,1] = PR[GP1:90,1] + 36.386;
   1:  PR[GP1:91,2] = PR[GP1:90,2] + 13.093;
   1:L PR[91] R[100]mm/sec CNT100;
   1:  PR[GP1:91,1] = PR[GP1:90,1] + 32.834;
   1:  PR[GP1:91,2] = PR[GP1:90,2] + 15.855;
   1:L PR[91] R[100]mm/sec CNT100;
   1:  PR[GP1:91,1] = PR[GP1:90,1] + 32.224;
   1:  PR[GP1:91,2] = PR[GP1:90,2] + 16.194;
   1:L PR[91] R[100]mm/sec CNT100;
   1:  PR[GP1:91,1] = PR[GP1:90,1] + 28.640;
   1:  PR[GP1:91,2] = PR[GP1:90,2] + 17.701;
   1:L PR[91] R[100]mm/sec CNT100;
   1:  PR[GP1:91,1] = PR[GP1:90,1] + 28.082;
   1:  PR[GP1:91,2] = PR[GP1:90,2] + 17.901;
   1:L PR[91] R[100]mm/sec CNT100;
   1:  PR[GP1:91,1] = PR[GP1:90,1] + 27.489;
   1:  PR[GP1:91,2] = PR[GP1:90,2] + 18.008;
   1:L PR[91] R[100]mm/sec CNT100;
   1:  PR[GP1:91,1] = PR[GP1:90,1] + 23.458;
   1:  PR[GP1:91,2] = PR[GP1:90,2] + 18.571;
   1:L PR[91] R[100]mm/sec CNT100;
   1:  PR[GP1:91,1] = PR[GP1:90,1] + 23.081;
   1:  PR[GP1:91,2] = PR[GP1:90,2] + 18.576;
   1:L PR[91] R[100]mm/sec CNT100;
   1:  PR[GP1:91,1] = PR[GP1:90,1] + 22.600;
   1:  PR[GP1:91,2] = PR[GP1:90,2] + 18.505;
   1:L PR[91] R[100]mm/sec CNT100;
   1:  PR[GP1:91,1] = PR[GP1:90,1] + 18.360;
   1:  PR[GP1:91,2] = PR[GP1:90,2] + 17.995;
   1:L PR[91] R[100]mm/sec CNT100;
   1:  PR[GP1:91,1] = PR[GP1:90,1] + 18.165;
   1:  PR[GP1:91,2] = PR[GP1:90,2] + 17.932;
   1:L PR[91] R[100]mm/sec CNT100;
   1:  PR[GP1:91,1] = PR[GP1:90,1] + 13.805;
   1:  PR[GP1:91,2] = PR[GP1:90,2] + 16.187;
   1:L PR[91] R[100]mm/sec CNT100;
   1:  PR[GP1:91,1] = PR[GP1:90,1] + 13.802;
   1:  PR[GP1:91,2] = PR[GP1:90,2] + 16.185;
   1:L PR[91] R[100]mm/sec CNT100;
   1:  PR[GP1:91,1] = PR[GP1:90,1] + 9.831;
   1:  PR[GP1:91,2] = PR[GP1:90,2] + 13.230;
   1:L PR[91] R[100]mm/sec CNT100;
   1:  PR[GP1:91,1] = PR[GP1:90,1] + 6.761;
   1:  PR[GP1:91,2] = PR[GP1:90,2] + 9.412;
   1:L PR[91] R[100]mm/sec CNT100;
   1:  PR[GP1:91,1] = PR[GP1:90,1] + 6.710;
   1:  PR[GP1:91,2] = PR[GP1:90,2] + 9.318;
   1:L PR[91] R[100]mm/sec CNT100;
   1:  PR[GP1:91,1] = PR[GP1:90,1] + 4.686;
   1:  PR[GP1:91,2] = PR[GP1:90,2] + 4.710;
   1:L PR[91] R[100]mm/sec CNT100;
   1:  PR[GP1:91,1] = PR[GP1:90,1] + 4.353;
   1:  PR[GP1:91,2] = PR[GP1:90,2] + 4.275;
   1:L PR[91] R[100]mm/sec CNT100;
   1:  PR[GP1:91,1] = PR[GP1:90,1] + 4.239;
   1:  PR[GP1:91,2] = PR[GP1:90,2] + 4.179;
   1:L PR[91] R[100]mm/sec CNT100;
   1:  PR[GP1:91,1] = PR[GP1:90,1] + 4.149;
   1:  PR[GP1:91,2] = PR[GP1:90,2] + 4.043;
   1:L PR[91] R[100]mm/sec CNT100;
   1:  PR[GP1:91,1] = PR[GP1:90,1] + 3.767;
   1:  PR[GP1:91,2] = PR[GP1:90,2] + 3.545;
   1:L PR[91] R[100]mm/sec CNT100;
   1:  PR[GP1:91,1] = PR[GP1:90,1] + 2.802;
   1:  PR[GP1:91,2] = PR[GP1:90,2] + 2.906;
   1:L PR[91] R[100]mm/sec CNT100;
   1:  PR[GP1:91,1] = PR[GP1:90,1] + 1.780;
   1:  PR[GP1:91,2] = PR[GP1:90,2] + 2.701;
   1:L PR[91] R[100]mm/sec CNT100;
   1:  PR[GP1:91,1] = PR[GP1:90,1] + -1.647;
   1:L PR[91] R[100]mm/sec CNT100;
   1:  PR[91] = PR[90];
   1:  PR[GP1:91,1] = PR[GP1:90,1] + -2.648;
   1:  PR[GP1:91,2] = PR[GP1:90,2] + 3.200;
   1:  PR[GP1:91,3] = PR[GP1:90,3] + 10.065;
   1:L PR[91] R[100]mm/sec CNT100;
   1:  PR[GP1:91,1] = PR[GP1:90,1] + -3.609;
   1:  PR[GP1:91,2] = PR[GP1:90,2] + 3.840;
   1:L PR[91] R[100]mm/sec CNT100;
   1:  PR[GP1:91,1] = PR[GP1:90,1] + -3.960;
   1:  PR[GP1:91,2] = PR[GP1:90,2] + 4.298;
   1:L PR[91] R[100]mm/sec CNT100;
   1:  PR[GP1:91,1] = PR[GP1:90,1] + -4.139;
   1:  PR[GP1:91,2] = PR[GP1:90,2] + 4.566;
   1:L PR[91] R[100]mm/sec CNT100;
   1:  PR[GP1:91,1] = PR[GP1:90,1] + -4.449;
   1:  PR[GP1:91,2] = PR[GP1:90,2] + 4.916;
   1:L PR[91] R[100]mm/sec CNT100;
   1:  PR[GP1:91,1] = PR[GP1:90,1] + -6.194;
   1:  PR[GP1:91,2] = PR[GP1:90,2] + 8.852;
   1:L PR[91] R[100]mm/sec CNT100;
   1:  PR[GP1:91,1] = PR[GP1:90,1] + -6.617;
   1:  PR[GP1:91,2] = PR[GP1:90,2] + 9.626;
   1:L PR[91] R[100]mm/sec CNT100;
   1:  PR[GP1:91,1] = PR[GP1:90,1] + -9.283;
   1:  PR[GP1:91,2] = PR[GP1:90,2] + 12.937;
   1:L PR[91] R[100]mm/sec CNT100;
   1:  PR[GP1:91,1] = PR[GP1:90,1] + -9.678;
   1:  PR[GP1:91,2] = PR[GP1:90,2] + 13.357;
   1:L PR[91] R[100]mm/sec CNT100;
   1:  PR[GP1:91,1] = PR[GP1:90,1] + -13.420;
   1:  PR[GP1:91,2] = PR[GP1:90,2] + 16.094;
   1:L PR[91] R[100]mm/sec CNT100;
   1:  PR[GP1:91,1] = PR[GP1:90,1] + -13.595;
   1:  PR[GP1:91,2] = PR[GP1:90,2] + 16.205;
   1:L PR[91] R[100]mm/sec CNT100;
   1:  PR[GP1:91,1] = PR[GP1:90,1] + -18.173;
   1:  PR[GP1:91,2] = PR[GP1:90,2] + 17.996;
   1:L PR[91] R[100]mm/sec CNT100;
   1:  PR[GP1:91,1] = PR[GP1:90,1] + -23.053;
   1:  PR[GP1:91,2] = PR[GP1:90,2] + 18.587;
   1:L PR[91] R[100]mm/sec CNT100;
   1:  PR[GP1:91,1] = PR[GP1:90,1] + -23.078;
   1:  PR[GP1:91,2] = PR[GP1:90,2] + 18.586;
   1:L PR[91] R[100]mm/sec CNT100;
   1:  PR[GP1:91,1] = PR[GP1:90,1] + -27.947;
   1:  PR[GP1:91,2] = PR[GP1:90,2] + 17.890;
   1:L PR[91] R[100]mm/sec CNT100;
   1:  PR[GP1:91,1] = PR[GP1:90,1] + -28.152;
   1:  PR[GP1:91,2] = PR[GP1:90,2] + 17.817;
   1:L PR[91] R[100]mm/sec CNT100;
   1:  PR[GP1:91,1] = PR[GP1:90,1] + -32.234;
   1:  PR[GP1:91,2] = PR[GP1:90,2] + 16.098;
   1:L PR[91] R[100]mm/sec CNT100;
   1:  PR[GP1:91,1] = PR[GP1:90,1] + -32.557;
   1:  PR[GP1:91,2] = PR[GP1:90,2] + 15.918;
   1:L PR[91] R[100]mm/sec CNT100;
   1:  PR[GP1:91,1] = PR[GP1:90,1] + -36.261;
   1:  PR[GP1:91,2] = PR[GP1:90,2] + 13.042;
   1:L PR[91] R[100]mm/sec CNT100;
   1:  PR[GP1:91,1] = PR[GP1:90,1] + -36.592;
   1:  PR[GP1:91,2] = PR[GP1:90,2] + 12.677;
   1:L PR[91] R[100]mm/sec CNT100;
   1:  PR[GP1:91,1] = PR[GP1:90,1] + -39.026;
   1:  PR[GP1:91,2] = PR[GP1:90,2] + 9.486;
   1:L PR[91] R[100]mm/sec CNT100;
   1:  PR[GP1:91,1] = PR[GP1:90,1] + -39.346;
   1:  PR[GP1:91,2] = PR[GP1:90,2] + 8.990;
   1:L PR[91] R[100]mm/sec CNT100;
   1:  PR[GP1:91,1] = PR[GP1:90,1] + -39.599;
   1:  PR[GP1:91,2] = PR[GP1:90,2] + 8.408;
   1:L PR[91] R[100]mm/sec CNT100;
   1:  PR[GP1:91,1] = PR[GP1:90,1] + -41.094;
   1:  PR[GP1:91,2] = PR[GP1:90,2] + 4.789;
   1:L PR[91] R[100]mm/sec CNT100;
   1:  PR[GP1:91,1] = PR[GP1:90,1] + -41.238;
   1:  PR[GP1:91,2] = PR[GP1:90,2] + 4.214;
   1:L PR[91] R[100]mm/sec CNT100;
   1:  PR[GP1:91,1] = PR[GP1:90,1] + -41.298;
   1:  PR[GP1:91,2] = PR[GP1:90,2] + 3.485;
   1:L PR[91] R[100]mm/sec CNT100;
   1:  PR[GP1:91,1] = PR[GP1:90,1] + -41.795;
   1:  PR[GP1:91,2] = PR[GP1:90,2] + -0.346;
   1:L PR[91] R[100]mm/sec CNT100;
   1:  PR[GP1:91,1] = PR[GP1:90,1] + -41.737;
   1:  PR[GP1:91,2] = PR[GP1:90,2] + -1.052;
   1:L PR[91] R[100]mm/sec CNT100;
   1:  PR[GP1:91,1] = PR[GP1:90,1] + -41.246;
   1:  PR[GP1:91,2] = PR[GP1:90,2] + -4.804;
   1:L PR[91] R[100]mm/sec CNT100;
   1:  PR[GP1:91,1] = PR[GP1:90,1] + -41.097;
   1:  PR[GP1:91,2] = PR[GP1:90,2] + -5.400;
   1:L PR[91] R[100]mm/sec CNT100;
   1:  PR[GP1:91,1] = PR[GP1:90,1] + -40.814;
   1:  PR[GP1:91,2] = PR[GP1:90,2] + -6.052;
   1:L PR[91] R[100]mm/sec CNT100;
   1:  PR[GP1:91,1] = PR[GP1:90,1] + -39.339;
   1:  PR[GP1:91,2] = PR[GP1:90,2] + -9.625;
   1:L PR[91] R[100]mm/sec CNT100;
   1:  PR[GP1:91,1] = PR[GP1:90,1] + -39.026;
   1:  PR[GP1:91,2] = PR[GP1:90,2] + -10.110;
   1:L PR[91] R[100]mm/sec CNT100;
   1:  PR[GP1:91,1] = PR[GP1:90,1] + -36.592;
   1:  PR[GP1:91,2] = PR[GP1:90,2] + -13.301;
   1:L PR[91] R[100]mm/sec CNT100;
   1:  PR[GP1:91,1] = PR[GP1:90,1] + -36.261;
   1:  PR[GP1:91,2] = PR[GP1:90,2] + -13.666;
   1:L PR[91] R[100]mm/sec CNT100;
   1:  PR[GP1:91,1] = PR[GP1:90,1] + -32.558;
   1:  PR[GP1:91,2] = PR[GP1:90,2] + -16.542;
   1:L PR[91] R[100]mm/sec CNT100;
   1:  PR[GP1:91,1] = PR[GP1:90,1] + -32.234;
   1:  PR[GP1:91,2] = PR[GP1:90,2] + -16.722;
   1:L PR[91] R[100]mm/sec CNT100;
   1:  PR[GP1:91,1] = PR[GP1:90,1] + -28.153;
   1:  PR[GP1:91,2] = PR[GP1:90,2] + -18.440;
   1:L PR[91] R[100]mm/sec CNT100;
   1:  PR[GP1:91,1] = PR[GP1:90,1] + -27.922;
   1:  PR[GP1:91,2] = PR[GP1:90,2] + -18.523;
   1:L PR[91] R[100]mm/sec CNT100;
   1:  PR[GP1:91,1] = PR[GP1:90,1] + -27.670;
   1:  PR[GP1:91,2] = PR[GP1:90,2] + -18.568;
   1:L PR[91] R[100]mm/sec CNT100;
   1:  PR[GP1:91,1] = PR[GP1:90,1] + -23.081;
   1:  PR[GP1:91,2] = PR[GP1:90,2] + -19.210;
   1:L PR[91] R[100]mm/sec CNT100;
   1:  PR[GP1:91,1] = PR[GP1:90,1] + -23.054;
   1:  PR[GP1:91,2] = PR[GP1:90,2] + -19.211;
   1:L PR[91] R[100]mm/sec CNT100;
   1:  PR[GP1:91,1] = PR[GP1:90,1] + -18.176;
   1:  PR[GP1:91,2] = PR[GP1:90,2] + -18.621;
   1:L PR[91] R[100]mm/sec CNT100;
   1:  PR[GP1:91,1] = PR[GP1:90,1] + -13.596;
   1:  PR[GP1:91,2] = PR[GP1:90,2] + -16.829;
   1:L PR[91] R[100]mm/sec CNT100;
   1:  PR[GP1:91,1] = PR[GP1:90,1] + -13.421;
   1:  PR[GP1:91,2] = PR[GP1:90,2] + -16.718;
   1:L PR[91] R[100]mm/sec CNT100;
   1:  PR[GP1:91,1] = PR[GP1:90,1] + -9.678;
   1:  PR[GP1:91,2] = PR[GP1:90,2] + -13.981;
   1:L PR[91] R[100]mm/sec CNT100;
   1:  PR[GP1:91,1] = PR[GP1:90,1] + -9.284;
   1:  PR[GP1:91,2] = PR[GP1:90,2] + -13.562;
   1:L PR[91] R[100]mm/sec CNT100;
   1:  PR[GP1:91,1] = PR[GP1:90,1] + -6.617;
   1:  PR[GP1:91,2] = PR[GP1:90,2] + -10.251;
   1:L PR[91] R[100]mm/sec CNT100;
   1:  PR[GP1:91,1] = PR[GP1:90,1] + -6.196;
   1:  PR[GP1:91,2] = PR[GP1:90,2] + -9.479;
   1:L PR[91] R[100]mm/sec CNT100;
   1:  PR[GP1:91,1] = PR[GP1:90,1] + -4.451;
   1:  PR[GP1:91,2] = PR[GP1:90,2] + -5.529;
   1:L PR[91] R[100]mm/sec CNT100;
   1:  PR[GP1:91,1] = PR[GP1:90,1] + -4.132;
   1:  PR[GP1:91,2] = PR[GP1:90,2] + -5.180;
   1:L PR[91] R[100]mm/sec CNT100;
   1:  PR[GP1:91,1] = PR[GP1:90,1] + -3.960;
   1:  PR[GP1:91,2] = PR[GP1:90,2] + -4.922;
   1:L PR[91] R[100]mm/sec CNT100;
   1:  PR[GP1:91,1] = PR[GP1:90,1] + -3.608;
   1:  PR[GP1:91,2] = PR[GP1:90,2] + -4.464;
   1:L PR[91] R[100]mm/sec CNT100;
   1:  PR[GP1:91,1] = PR[GP1:90,1] + -2.646;
   1:  PR[GP1:91,2] = PR[GP1:90,2] + -3.822;
   1:L PR[91] R[100]mm/sec CNT100;
   1:  PR[GP1:91,1] = PR[GP1:90,1] + -1.632;
   1:  PR[GP1:91,2] = PR[GP1:90,2] + -3.613;
   1:L PR[91] R[100]mm/sec CNT100;
   1:  PR[GP1:91,1] = PR[GP1:90,1] + 1.778;
   1:L PR[91] R[100]mm/sec CNT100;
   1:  PR[GP1:91,1] = PR[GP1:90,1] + 2.799;
   1:  PR[GP1:91,2] = PR[GP1:90,2] + -3.821;
   1:L PR[91] R[100]mm/sec CNT100;
   1:  PR[GP1:91,1] = PR[GP1:90,1] + 3.763;
   1:  PR[GP1:91,2] = PR[GP1:90,2] + -4.463;
   1:L PR[91] R[100]mm/sec CNT100;
   1:  PR[GP1:91,1] = PR[GP1:90,1] + 4.115;
   1:  PR[GP1:91,2] = PR[GP1:90,2] + -4.921;
   1:L PR[91] R[100]mm/sec CNT100;
   1:  PR[GP1:91,1] = PR[GP1:90,1] + 4.293;
   1:  PR[GP1:91,2] = PR[GP1:90,2] + -5.188;
   1:L PR[91] R[100]mm/sec CNT100;
   1:  PR[GP1:91,1] = PR[GP1:90,1] + 4.604;
   1:  PR[GP1:91,2] = PR[GP1:90,2] + -5.539;
   1:L PR[91] R[100]mm/sec CNT100;
   1:  PR[GP1:91,1] = PR[GP1:90,1] + 6.348;
   1:  PR[GP1:91,2] = PR[GP1:90,2] + -9.470;
   1:L PR[91] R[100]mm/sec CNT100;
   1:  PR[GP1:91,1] = PR[GP1:90,1] + 6.772;
   1:  PR[GP1:91,2] = PR[GP1:90,2] + -10.246;
   1:L PR[91] R[100]mm/sec CNT100;
   1:  PR[GP1:91,1] = PR[GP1:90,1] + 9.439;
   1:  PR[GP1:91,2] = PR[GP1:90,2] + -13.560;
   1:L PR[91] R[100]mm/sec CNT100;
   1:  PR[GP1:91,1] = PR[GP1:90,1] + 9.834;
   1:  PR[GP1:91,2] = PR[GP1:90,2] + -13.980;
   1:L PR[91] R[100]mm/sec CNT100;
   1:  PR[GP1:91,1] = PR[GP1:90,1] + 13.575;
   1:  PR[GP1:91,2] = PR[GP1:90,2] + -16.718;
   1:L PR[91] R[100]mm/sec CNT100;
   1:  PR[GP1:91,1] = PR[GP1:90,1] + 13.751;
   1:  PR[GP1:91,2] = PR[GP1:90,2] + -16.829;
   1:L PR[91] R[100]mm/sec CNT100;
   1:  PR[GP1:91,1] = PR[GP1:90,1] + 18.329;
   1:  PR[GP1:91,2] = PR[GP1:90,2] + -18.619;
   1:L PR[91] R[100]mm/sec CNT100;
   1:  PR[GP1:91,1] = PR[GP1:90,1] + 23.210;
   1:  PR[GP1:91,2] = PR[GP1:90,2] + -19.211;
   1:L PR[91] R[100]mm/sec CNT100;
   1:  PR[GP1:91,1] = PR[GP1:90,1] + 23.234;
   1:  PR[GP1:91,2] = PR[GP1:90,2] + -19.210;
   1:L PR[91] R[100]mm/sec CNT100;
   1:  PR[GP1:91,1] = PR[GP1:90,1] + 28.103;
   1:  PR[GP1:91,2] = PR[GP1:90,2] + -18.514;
   1:L PR[91] R[100]mm/sec CNT100;
   1:  PR[GP1:91,1] = PR[GP1:90,1] + 28.308;
   1:  PR[GP1:91,2] = PR[GP1:90,2] + -18.440;
   1:L PR[91] R[100]mm/sec CNT100;
   1:  PR[GP1:91,1] = PR[GP1:90,1] + 32.390;
   1:  PR[GP1:91,2] = PR[GP1:90,2] + -16.722;
   1:L PR[91] R[100]mm/sec CNT100;
   1:  PR[GP1:91,1] = PR[GP1:90,1] + 32.714;
   1:  PR[GP1:91,2] = PR[GP1:90,2] + -16.543;
   1:L PR[91] R[100]mm/sec CNT100;
   1:  PR[GP1:91,1] = PR[GP1:90,1] + 36.417;
   1:  PR[GP1:91,2] = PR[GP1:90,2] + -13.667;
   1:L PR[91] R[100]mm/sec CNT100;
   1:  PR[GP1:91,1] = PR[GP1:90,1] + 36.748;
   1:  PR[GP1:91,2] = PR[GP1:90,2] + -13.302;
   1:L PR[91] R[100]mm/sec CNT100;
   1:  PR[GP1:91,1] = PR[GP1:90,1] + 39.183;
   1:  PR[GP1:91,2] = PR[GP1:90,2] + -10.109;
   1:L PR[91] R[100]mm/sec CNT100;
   1:  PR[GP1:91,1] = PR[GP1:90,1] + 39.503;
   1:  PR[GP1:91,2] = PR[GP1:90,2] + -9.613;
   1:L PR[91] R[100]mm/sec CNT100;
   1:  PR[GP1:91,1] = PR[GP1:90,1] + 39.755;
   1:  PR[GP1:91,2] = PR[GP1:90,2] + -9.031;
   1:L PR[91] R[100]mm/sec CNT100;
   1:  PR[GP1:91,1] = PR[GP1:90,1] + 41.251;
   1:  PR[GP1:91,2] = PR[GP1:90,2] + -5.415;
   1:L PR[91] R[100]mm/sec CNT100;
   1:  PR[GP1:91,1] = PR[GP1:90,1] + 41.395;
   1:  PR[GP1:91,2] = PR[GP1:90,2] + -4.841;
   1:L PR[91] R[100]mm/sec CNT100;
   1:  PR[GP1:91,1] = PR[GP1:90,1] + 41.454;
   1:  PR[GP1:91,2] = PR[GP1:90,2] + -4.112;
   1:L PR[91] R[100]mm/sec CNT100;
   1:  PR[GP1:91,1] = PR[GP1:90,1] + 41.951;
   1:  PR[GP1:91,2] = PR[GP1:90,2] + -0.278;
   1:L PR[91] R[100]mm/sec CNT100;
   1:  PR[GP1:91,1] = PR[GP1:90,1] + 41.894;
   1:  PR[GP1:91,2] = PR[GP1:90,2] + 0.428;
   1:L PR[91] R[100]mm/sec CNT100;
   1:  PR[GP1:91,1] = PR[GP1:90,1] + 41.403;
   1:  PR[GP1:91,2] = PR[GP1:90,2] + 4.184;
   1:L PR[91] R[100]mm/sec CNT100;
   1:  PR[GP1:91,1] = PR[GP1:90,1] + 41.254;
   1:  PR[GP1:91,2] = PR[GP1:90,2] + 4.780;
   1:L PR[91] R[100]mm/sec CNT100;
   1:  PR[GP1:91,1] = PR[GP1:90,1] + 40.971;
   1:  PR[GP1:91,2] = PR[GP1:90,2] + 5.431;
   1:L PR[91] R[100]mm/sec CNT100;
   1:  PR[GP1:91,1] = PR[GP1:90,1] + 39.495;
   1:  PR[GP1:91,2] = PR[GP1:90,2] + 9.001;
   1:L PR[91] R[100]mm/sec CNT100;
   1:  PR[GP1:91,1] = PR[GP1:90,1] + 39.182;
   1:  PR[GP1:91,2] = PR[GP1:90,2] + 9.487;
   1:L PR[91] R[100]mm/sec CNT100;
   1:  PR[GP1:91,1] = PR[GP1:90,1] + 36.746;
   1:  PR[GP1:91,2] = PR[GP1:90,2] + 12.680;
   1:L PR[91] R[100]mm/sec CNT100;
   1:  PR[GP1:91,1] = PR[GP1:90,1] + 36.416;
   1:  PR[GP1:91,2] = PR[GP1:90,2] + 13.044;
   1:L PR[91] R[100]mm/sec CNT100;
   1:  PR[GP1:91,1] = PR[GP1:90,1] + 32.711;
   1:  PR[GP1:91,2] = PR[GP1:90,2] + 15.921;
   1:L PR[91] R[100]mm/sec CNT100;
   1:  PR[GP1:91,1] = PR[GP1:90,1] + 32.387;
   1:  PR[GP1:91,2] = PR[GP1:90,2] + 16.100;
   1:L PR[91] R[100]mm/sec CNT100;
   1:  PR[GP1:91,1] = PR[GP1:90,1] + 28.303;
   1:  PR[GP1:91,2] = PR[GP1:90,2] + 17.818;
   1:L PR[91] R[100]mm/sec CNT100;
   1:  PR[GP1:91,1] = PR[GP1:90,1] + 28.073;
   1:  PR[GP1:91,2] = PR[GP1:90,2] + 17.900;
   1:L PR[91] R[100]mm/sec CNT100;
   1:  PR[GP1:91,1] = PR[GP1:90,1] + 27.822;
   1:  PR[GP1:91,2] = PR[GP1:90,2] + 17.946;
   1:L PR[91] R[100]mm/sec CNT100;
   1:  PR[GP1:91,1] = PR[GP1:90,1] + 23.230;
   1:  PR[GP1:91,2] = PR[GP1:90,2] + 18.586;
   1:L PR[91] R[100]mm/sec CNT100;
   1:  PR[GP1:91,1] = PR[GP1:90,1] + 23.203;
   1:  PR[GP1:91,2] = PR[GP1:90,2] + 18.587;
   1:L PR[91] R[100]mm/sec CNT100;
   1:  PR[GP1:91,1] = PR[GP1:90,1] + 18.324;
   1:  PR[GP1:91,2] = PR[GP1:90,2] + 17.994;
   1:L PR[91] R[100]mm/sec CNT100;
   1:  PR[GP1:91,1] = PR[GP1:90,1] + 13.744;
   1:  PR[GP1:91,2] = PR[GP1:90,2] + 16.201;
   1:L PR[91] R[100]mm/sec CNT100;
   1:  PR[GP1:91,1] = PR[GP1:90,1] + 13.568;
   1:  PR[GP1:91,2] = PR[GP1:90,2] + 16.090;
   1:L PR[91] R[100]mm/sec CNT100;
   1:  PR[GP1:91,1] = PR[GP1:90,1] + 9.828;
   1:  PR[GP1:91,2] = PR[GP1:90,2] + 13.351;
   1:L PR[91] R[100]mm/sec CNT100;
   1:  PR[GP1:91,1] = PR[GP1:90,1] + 9.434;
   1:  PR[GP1:91,2] = PR[GP1:90,2] + 12.930;
   1:L PR[91] R[100]mm/sec CNT100;
   1:  PR[GP1:91,1] = PR[GP1:90,1] + 6.768;
   1:  PR[GP1:91,2] = PR[GP1:90,2] + 9.615;
   1:L PR[91] R[100]mm/sec CNT100;
   1:  PR[GP1:91,1] = PR[GP1:90,1] + 6.347;
   1:  PR[GP1:91,2] = PR[GP1:90,2] + 8.847;
   1:L PR[91] R[100]mm/sec CNT100;
   1:  PR[GP1:91,1] = PR[GP1:90,1] + 5.505;
   1:  PR[GP1:91,2] = PR[GP1:90,2] + 6.934;
   1:L PR[91] R[100]mm/sec CNT100;
   1:  PR[GP1:91,1] = PR[GP1:90,1] + 6.114;
   1:  PR[GP1:91,2] = PR[GP1:90,2] + 6.873;
   1:L PR[91] R[100]mm/sec CNT100;
   1:  PR[GP1:91,1] = PR[GP1:90,1] + 4.373;
   1:  PR[GP1:91,2] = PR[GP1:90,2] + 4.594;
   1:L PR[91] R[100]mm/sec CNT100;
   1:  PR[GP1:91,1] = PR[GP1:90,1] + 4.235;
   1:  PR[GP1:91,2] = PR[GP1:90,2] + 4.478;
   1:L PR[91] R[100]mm/sec CNT100;
   1:  PR[GP1:91,1] = PR[GP1:90,1] + 4.116;
   1:  PR[GP1:91,2] = PR[GP1:90,2] + 4.299;
   1:L PR[91] R[100]mm/sec CNT100;
   1:  PR[GP1:91,1] = PR[GP1:90,1] + 3.765;
   1:  PR[GP1:91,2] = PR[GP1:90,2] + 3.841;
   1:L PR[91] R[100]mm/sec CNT100;
   1:  PR[GP1:91,1] = PR[GP1:90,1] + 2.800;
   1:  PR[GP1:91,2] = PR[GP1:90,2] + 3.197;
   1:L PR[91] R[100]mm/sec CNT100;
   1:  PR[GP1:91,1] = PR[GP1:90,1] + 1.771;
   1:  PR[GP1:91,2] = PR[GP1:90,2] + 2.989;
   1:L PR[91] R[100]mm/sec CNT100;
   1:  PR[GP1:91,1] = PR[GP1:90,1] + -1.643;
   1:L PR[91] R[100]mm/sec CNT100;
   1:  PR[91] = PR[90];
   1:  PR[GP1:91,1] = PR[GP1:90,1] + -2.646;
   1:  PR[GP1:91,2] = PR[GP1:90,2] + 3.491;
   1:  PR[GP1:91,3] = PR[GP1:90,3] + 10.675;
   1:L PR[91] R[100]mm/sec CNT100;
   1:  PR[GP1:91,1] = PR[GP1:90,1] + -3.607;
   1:  PR[GP1:91,2] = PR[GP1:90,2] + 4.136;
   1:L PR[91] R[100]mm/sec CNT100;
   1:  PR[GP1:91,1] = PR[GP1:90,1] + -3.927;
   1:  PR[GP1:91,2] = PR[GP1:90,2] + 4.554;
   1:L PR[91] R[100]mm/sec CNT100;
   1:  PR[GP1:91,1] = PR[GP1:90,1] + -4.079;
   1:  PR[GP1:91,2] = PR[GP1:90,2] + 4.781;
   1:L PR[91] R[100]mm/sec CNT100;
   1:  PR[GP1:91,1] = PR[GP1:90,1] + -4.420;
   1:  PR[GP1:91,2] = PR[GP1:90,2] + 5.192;
   1:L PR[91] R[100]mm/sec CNT100;
   1:  PR[GP1:91,1] = PR[GP1:90,1] + -5.830;
   1:  PR[GP1:91,2] = PR[GP1:90,2] + 8.376;
   1:L PR[91] R[100]mm/sec CNT100;
   1:  PR[GP1:91,1] = PR[GP1:90,1] + -6.622;
   1:  PR[GP1:91,2] = PR[GP1:90,2] + 9.828;
   1:L PR[91] R[100]mm/sec CNT100;
   1:  PR[GP1:91,1] = PR[GP1:90,1] + -8.804;
   1:  PR[GP1:91,2] = PR[GP1:90,2] + 12.536;
   1:L PR[91] R[100]mm/sec CNT100;
   1:  PR[GP1:91,1] = PR[GP1:90,1] + -9.711;
   1:  PR[GP1:91,2] = PR[GP1:90,2] + 13.501;
   1:L PR[91] R[100]mm/sec CNT100;
   1:  PR[GP1:91,1] = PR[GP1:90,1] + -12.855;
   1:  PR[GP1:91,2] = PR[GP1:90,2] + 15.801;
   1:L PR[91] R[100]mm/sec CNT100;
   1:  PR[GP1:91,1] = PR[GP1:90,1] + -13.637;
   1:  PR[GP1:91,2] = PR[GP1:90,2] + 16.296;
   1:L PR[91] R[100]mm/sec CNT100;
   1:  PR[GP1:91,1] = PR[GP1:90,1] + -17.692;
   1:  PR[GP1:91,2] = PR[GP1:90,2] + 17.882;
   1:L PR[91] R[100]mm/sec CNT100;
   1:  PR[GP1:91,1] = PR[GP1:90,1] + -18.166;
   1:  PR[GP1:91,2] = PR[GP1:90,2] + 18.036;
   1:L PR[91] R[100]mm/sec CNT100;
   1:  PR[GP1:91,1] = PR[GP1:90,1] + -22.930;
   1:  PR[GP1:91,2] = PR[GP1:90,2] + 18.587;
   1:L PR[91] R[100]mm/sec CNT100;
   1:  PR[GP1:91,1] = PR[GP1:90,1] + -23.014;
   1:  PR[GP1:91,2] = PR[GP1:90,2] + 18.592;
   1:L PR[91] R[100]mm/sec CNT100;
   1:  PR[GP1:91,1] = PR[GP1:90,1] + -27.899;
   1:  PR[GP1:91,2] = PR[GP1:90,2] + 17.895;
   1:L PR[91] R[100]mm/sec CNT100;
   1:  PR[GP1:91,1] = PR[GP1:90,1] + -32.398;
   1:  PR[GP1:91,2] = PR[GP1:90,2] + 16.004;
   1:L PR[91] R[100]mm/sec CNT100;
   1:  PR[GP1:91,1] = PR[GP1:90,1] + -32.434;
   1:  PR[GP1:91,2] = PR[GP1:90,2] + 15.984;
   1:L PR[91] R[100]mm/sec CNT100;
   1:  PR[GP1:91,1] = PR[GP1:90,1] + -36.291;
   1:  PR[GP1:91,2] = PR[GP1:90,2] + 12.993;
   1:L PR[91] R[100]mm/sec CNT100;
   1:  PR[GP1:91,1] = PR[GP1:90,1] + -36.410;
   1:  PR[GP1:91,2] = PR[GP1:90,2] + 12.862;
   1:L PR[91] R[100]mm/sec CNT100;
   1:  PR[GP1:91,1] = PR[GP1:90,1] + -39.143;
   1:  PR[GP1:91,2] = PR[GP1:90,2] + 9.279;
   1:L PR[91] R[100]mm/sec CNT100;
   1:  PR[GP1:91,1] = PR[GP1:90,1] + -39.292;
   1:  PR[GP1:91,2] = PR[GP1:90,2] + 9.049;
   1:L PR[91] R[100]mm/sec CNT100;
   1:  PR[GP1:91,1] = PR[GP1:90,1] + -41.109;
   1:  PR[GP1:91,2] = PR[GP1:90,2] + 4.671;
   1:L PR[91] R[100]mm/sec CNT100;
   1:  PR[GP1:91,1] = PR[GP1:90,1] + -41.180;
   1:  PR[GP1:91,2] = PR[GP1:90,2] + 4.387;
   1:L PR[91] R[100]mm/sec CNT100;
   1:  PR[GP1:91,1] = PR[GP1:90,1] + -41.215;
   1:  PR[GP1:91,2] = PR[GP1:90,2] + 3.955;
   1:L PR[91] R[100]mm/sec CNT100;
   1:  PR[GP1:91,1] = PR[GP1:90,1] + -41.773;
   1:  PR[GP1:91,2] = PR[GP1:90,2] + -0.346;
   1:L PR[91] R[100]mm/sec CNT100;
   1:  PR[GP1:91,1] = PR[GP1:90,1] + -41.739;
   1:  PR[GP1:91,2] = PR[GP1:90,2] + -0.764;
   1:L PR[91] R[100]mm/sec CNT100;
   1:  PR[GP1:91,1] = PR[GP1:90,1] + -41.188;
   1:  PR[GP1:91,2] = PR[GP1:90,2] + -4.977;
   1:L PR[91] R[100]mm/sec CNT100;
   1:  PR[GP1:91,1] = PR[GP1:90,1] + -41.109;
   1:  PR[GP1:91,2] = PR[GP1:90,2] + -5.295;
   1:L PR[91] R[100]mm/sec CNT100;
   1:  PR[GP1:91,1] = PR[GP1:90,1] + -39.292;
   1:  PR[GP1:91,2] = PR[GP1:90,2] + -9.672;
   1:L PR[91] R[100]mm/sec CNT100;
   1:  PR[GP1:91,1] = PR[GP1:90,1] + -39.143;
   1:  PR[GP1:91,2] = PR[GP1:90,2] + -9.903;
   1:L PR[91] R[100]mm/sec CNT100;
   1:  PR[GP1:91,1] = PR[GP1:90,1] + -36.411;
   1:  PR[GP1:91,2] = PR[GP1:90,2] + -13.486;
   1:L PR[91] R[100]mm/sec CNT100;
   1:  PR[GP1:91,1] = PR[GP1:90,1] + -36.291;
   1:  PR[GP1:91,2] = PR[GP1:90,2] + -13.617;
   1:L PR[91] R[100]mm/sec CNT100;
   1:  PR[GP1:91,1] = PR[GP1:90,1] + -32.434;
   1:  PR[GP1:91,2] = PR[GP1:90,2] + -16.607;
   1:L PR[91] R[100]mm/sec CNT100;
   1:  PR[GP1:91,1] = PR[GP1:90,1] + -32.398;
   1:  PR[GP1:91,2] = PR[GP1:90,2] + -16.628;
   1:L PR[91] R[100]mm/sec CNT100;
   1:  PR[GP1:91,1] = PR[GP1:90,1] + -27.900;
   1:  PR[GP1:91,2] = PR[GP1:90,2] + -18.519;
   1:L PR[91] R[100]mm/sec CNT100;
   1:  PR[GP1:91,1] = PR[GP1:90,1] + -23.014;
   1:  PR[GP1:91,2] = PR[GP1:90,2] + -19.216;
   1:L PR[91] R[100]mm/sec CNT100;
   1:  PR[GP1:91,1] = PR[GP1:90,1] + -22.930;
   1:  PR[GP1:91,2] = PR[GP1:90,2] + -19.211;
   1:L PR[91] R[100]mm/sec CNT100;
   1:  PR[GP1:91,1] = PR[GP1:90,1] + -18.166;
   1:  PR[GP1:91,2] = PR[GP1:90,2] + -18.660;
   1:L PR[91] R[100]mm/sec CNT100;
   1:  PR[GP1:91,1] = PR[GP1:90,1] + -17.693;
   1:  PR[GP1:91,2] = PR[GP1:90,2] + -18.506;
   1:L PR[91] R[100]mm/sec CNT100;
   1:  PR[GP1:91,1] = PR[GP1:90,1] + -13.637;
   1:  PR[GP1:91,2] = PR[GP1:90,2] + -16.920;
   1:L PR[91] R[100]mm/sec CNT100;
   1:  PR[GP1:91,1] = PR[GP1:90,1] + -12.855;
   1:  PR[GP1:91,2] = PR[GP1:90,2] + -16.425;
   1:L PR[91] R[100]mm/sec CNT100;
   1:  PR[GP1:91,1] = PR[GP1:90,1] + -9.711;
   1:  PR[GP1:91,2] = PR[GP1:90,2] + -14.126;
   1:L PR[91] R[100]mm/sec CNT100;
   1:  PR[GP1:91,1] = PR[GP1:90,1] + -8.804;
   1:  PR[GP1:91,2] = PR[GP1:90,2] + -13.160;
   1:L PR[91] R[100]mm/sec CNT100;
   1:  PR[GP1:91,1] = PR[GP1:90,1] + -6.622;
   1:  PR[GP1:91,2] = PR[GP1:90,2] + -10.452;
   1:L PR[91] R[100]mm/sec CNT100;
   1:  PR[GP1:91,1] = PR[GP1:90,1] + -5.831;
   1:  PR[GP1:91,2] = PR[GP1:90,2] + -9.003;
   1:L PR[91] R[100]mm/sec CNT100;
   1:  PR[GP1:91,1] = PR[GP1:90,1] + -4.407;
   1:  PR[GP1:91,2] = PR[GP1:90,2] + -5.779;
   1:L PR[91] R[100]mm/sec CNT100;
   1:  PR[GP1:91,1] = PR[GP1:90,1] + -4.125;
   1:  PR[GP1:91,2] = PR[GP1:90,2] + -5.475;
   1:L PR[91] R[100]mm/sec CNT100;
   1:  PR[GP1:91,1] = PR[GP1:90,1] + -3.927;
   1:  PR[GP1:91,2] = PR[GP1:90,2] + -5.178;
   1:L PR[91] R[100]mm/sec CNT100;
   1:  PR[GP1:91,1] = PR[GP1:90,1] + -3.606;
   1:  PR[GP1:91,2] = PR[GP1:90,2] + -4.760;
   1:L PR[91] R[100]mm/sec CNT100;
   1:  PR[GP1:91,1] = PR[GP1:90,1] + -2.644;
   1:  PR[GP1:91,2] = PR[GP1:90,2] + -4.113;
   1:L PR[91] R[100]mm/sec CNT100;
   1:  PR[GP1:91,1] = PR[GP1:90,1] + -1.626;
   1:  PR[GP1:91,2] = PR[GP1:90,2] + -3.902;
   1:L PR[91] R[100]mm/sec CNT100;
   1:  PR[GP1:91,1] = PR[GP1:90,1] + 1.770;
   1:L PR[91] R[100]mm/sec CNT100;
   1:  PR[GP1:91,1] = PR[GP1:90,1] + 2.796;
   1:  PR[GP1:91,2] = PR[GP1:90,2] + -4.112;
   1:L PR[91] R[100]mm/sec CNT100;
   1:  PR[GP1:91,1] = PR[GP1:90,1] + 3.760;
   1:  PR[GP1:91,2] = PR[GP1:90,2] + -4.758;
   1:L PR[91] R[100]mm/sec CNT100;
   1:  PR[GP1:91,1] = PR[GP1:90,1] + 4.082;
   1:  PR[GP1:91,2] = PR[GP1:90,2] + -5.177;
   1:L PR[91] R[100]mm/sec CNT100;
   1:  PR[GP1:91,1] = PR[GP1:90,1] + 4.285;
   1:  PR[GP1:91,2] = PR[GP1:90,2] + -5.482;
   1:L PR[91] R[100]mm/sec CNT100;
   1:  PR[GP1:91,1] = PR[GP1:90,1] + 4.560;
   1:  PR[GP1:91,2] = PR[GP1:90,2] + -5.788;
   1:L PR[91] R[100]mm/sec CNT100;
   1:  PR[GP1:91,1] = PR[GP1:90,1] + 5.983;
   1:  PR[GP1:91,2] = PR[GP1:90,2] + -8.992;
   1:L PR[91] R[100]mm/sec CNT100;
   1:  PR[GP1:91,1] = PR[GP1:90,1] + 6.777;
   1:  PR[GP1:91,2] = PR[GP1:90,2] + -10.446;
   1:L PR[91] R[100]mm/sec CNT100;
   1:  PR[GP1:91,1] = PR[GP1:90,1] + 8.959;
   1:  PR[GP1:91,2] = PR[GP1:90,2] + -13.157;
   1:L PR[91] R[100]mm/sec CNT100;
   1:  PR[GP1:91,1] = PR[GP1:90,1] + 9.866;
   1:  PR[GP1:91,2] = PR[GP1:90,2] + -14.125;
   1:L PR[91] R[100]mm/sec CNT100;
   1:  PR[GP1:91,1] = PR[GP1:90,1] + 13.010;
   1:  PR[GP1:91,2] = PR[GP1:90,2] + -16.425;
   1:L PR[91] R[100]mm/sec CNT100;
   1:  PR[GP1:91,1] = PR[GP1:90,1] + 13.792;
   1:  PR[GP1:91,2] = PR[GP1:90,2] + -16.919;
   1:L PR[91] R[100]mm/sec CNT100;
   1:  PR[GP1:91,1] = PR[GP1:90,1] + 17.848;
   1:  PR[GP1:91,2] = PR[GP1:90,2] + -18.506;
   1:L PR[91] R[100]mm/sec CNT100;
   1:  PR[GP1:91,1] = PR[GP1:90,1] + 18.321;
   1:  PR[GP1:91,2] = PR[GP1:90,2] + -18.660;
   1:L PR[91] R[100]mm/sec CNT100;
   1:  PR[GP1:91,1] = PR[GP1:90,1] + 23.086;
   1:  PR[GP1:91,2] = PR[GP1:90,2] + -19.211;
   1:L PR[91] R[100]mm/sec CNT100;
   1:  PR[GP1:91,1] = PR[GP1:90,1] + 23.170;
   1:  PR[GP1:91,2] = PR[GP1:90,2] + -19.216;
   1:L PR[91] R[100]mm/sec CNT100;
   1:  PR[GP1:91,1] = PR[GP1:90,1] + 28.055;
   1:  PR[GP1:91,2] = PR[GP1:90,2] + -18.519;
   1:L PR[91] R[100]mm/sec CNT100;
   1:  PR[GP1:91,1] = PR[GP1:90,1] + 32.554;
   1:  PR[GP1:91,2] = PR[GP1:90,2] + -16.628;
   1:L PR[91] R[100]mm/sec CNT100;
   1:  PR[GP1:91,1] = PR[GP1:90,1] + 32.590;
   1:  PR[GP1:91,2] = PR[GP1:90,2] + -16.608;
   1:L PR[91] R[100]mm/sec CNT100;
   1:  PR[GP1:91,1] = PR[GP1:90,1] + 36.448;
   1:  PR[GP1:91,2] = PR[GP1:90,2] + -13.618;
   1:L PR[91] R[100]mm/sec CNT100;
   1:  PR[GP1:91,1] = PR[GP1:90,1] + 36.567;
   1:  PR[GP1:91,2] = PR[GP1:90,2] + -13.486;
   1:L PR[91] R[100]mm/sec CNT100;
   1:  PR[GP1:91,1] = PR[GP1:90,1] + 39.300;
   1:  PR[GP1:91,2] = PR[GP1:90,2] + -9.902;
   1:L PR[91] R[100]mm/sec CNT100;
   1:  PR[GP1:91,1] = PR[GP1:90,1] + 39.449;
   1:  PR[GP1:91,2] = PR[GP1:90,2] + -9.671;
   1:L PR[91] R[100]mm/sec CNT100;
   1:  PR[GP1:91,1] = PR[GP1:90,1] + 41.266;
   1:  PR[GP1:91,2] = PR[GP1:90,2] + -5.298;
   1:L PR[91] R[100]mm/sec CNT100;
   1:  PR[GP1:91,1] = PR[GP1:90,1] + 41.337;
   1:  PR[GP1:91,2] = PR[GP1:90,2] + -5.014;
   1:L PR[91] R[100]mm/sec CNT100;
   1:  PR[GP1:91,1] = PR[GP1:90,1] + 41.372;
   1:  PR[GP1:91,2] = PR[GP1:90,2] + -4.582;
   1:L PR[91] R[100]mm/sec CNT100;
   1:  PR[GP1:91,1] = PR[GP1:90,1] + 41.930;
   1:  PR[GP1:91,2] = PR[GP1:90,2] + -0.278;
   1:L PR[91] R[100]mm/sec CNT100;
   1:  PR[GP1:91,1] = PR[GP1:90,1] + 41.896;
   1:  PR[GP1:91,2] = PR[GP1:90,2] + 0.140;
   1:L PR[91] R[100]mm/sec CNT100;
   1:  PR[GP1:91,1] = PR[GP1:90,1] + 41.345;
   1:  PR[GP1:91,2] = PR[GP1:90,2] + 4.357;
   1:L PR[91] R[100]mm/sec CNT100;
   1:  PR[GP1:91,1] = PR[GP1:90,1] + 41.265;
   1:  PR[GP1:91,2] = PR[GP1:90,2] + 4.675;
   1:L PR[91] R[100]mm/sec CNT100;
   1:  PR[GP1:91,1] = PR[GP1:90,1] + 39.448;
   1:  PR[GP1:91,2] = PR[GP1:90,2] + 9.049;
   1:L PR[91] R[100]mm/sec CNT100;
   1:  PR[GP1:91,1] = PR[GP1:90,1] + 39.299;
   1:  PR[GP1:91,2] = PR[GP1:90,2] + 9.280;
   1:L PR[91] R[100]mm/sec CNT100;
   1:  PR[GP1:91,1] = PR[GP1:90,1] + 36.565;
   1:  PR[GP1:91,2] = PR[GP1:90,2] + 12.864;
   1:L PR[91] R[100]mm/sec CNT100;
   1:  PR[GP1:91,1] = PR[GP1:90,1] + 36.445;
   1:  PR[GP1:91,2] = PR[GP1:90,2] + 12.996;
   1:L PR[91] R[100]mm/sec CNT100;
   1:  PR[GP1:91,1] = PR[GP1:90,1] + 32.587;
   1:  PR[GP1:91,2] = PR[GP1:90,2] + 15.986;
   1:L PR[91] R[100]mm/sec CNT100;
   1:  PR[GP1:91,1] = PR[GP1:90,1] + 32.551;
   1:  PR[GP1:91,2] = PR[GP1:90,2] + 16.006;
   1:L PR[91] R[100]mm/sec CNT100;
   1:  PR[GP1:91,1] = PR[GP1:90,1] + 28.050;
   1:  PR[GP1:91,2] = PR[GP1:90,2] + 17.896;
   1:L PR[91] R[100]mm/sec CNT100;
   1:  PR[GP1:91,1] = PR[GP1:90,1] + 23.163;
   1:  PR[GP1:91,2] = PR[GP1:90,2] + 18.592;
   1:L PR[91] R[100]mm/sec CNT100;
   1:  PR[GP1:91,1] = PR[GP1:90,1] + 23.079;
   1:  PR[GP1:91,2] = PR[GP1:90,2] + 18.587;
   1:L PR[91] R[100]mm/sec CNT100;
   1:  PR[GP1:91,1] = PR[GP1:90,1] + 18.315;
   1:  PR[GP1:91,2] = PR[GP1:90,2] + 18.034;
   1:L PR[91] R[100]mm/sec CNT100;
   1:  PR[GP1:91,1] = PR[GP1:90,1] + 17.841;
   1:  PR[GP1:91,2] = PR[GP1:90,2] + 17.880;
   1:L PR[91] R[100]mm/sec CNT100;
   1:  PR[GP1:91,1] = PR[GP1:90,1] + 13.786;
   1:  PR[GP1:91,2] = PR[GP1:90,2] + 16.292;
   1:L PR[91] R[100]mm/sec CNT100;
   1:  PR[GP1:91,1] = PR[GP1:90,1] + 13.004;
   1:  PR[GP1:91,2] = PR[GP1:90,2] + 15.798;
   1:L PR[91] R[100]mm/sec CNT100;
   1:  PR[GP1:91,1] = PR[GP1:90,1] + 9.862;
   1:  PR[GP1:91,2] = PR[GP1:90,2] + 13.497;
   1:L PR[91] R[100]mm/sec CNT100;
   1:  PR[GP1:91,1] = PR[GP1:90,1] + 8.955;
   1:  PR[GP1:91,2] = PR[GP1:90,2] + 12.530;
   1:L PR[91] R[100]mm/sec CNT100;
   1:  PR[GP1:91,1] = PR[GP1:90,1] + 6.774;
   1:  PR[GP1:91,2] = PR[GP1:90,2] + 9.817;
   1:L PR[91] R[100]mm/sec CNT100;
   1:  PR[GP1:91,1] = PR[GP1:90,1] + 5.985;
   1:  PR[GP1:91,2] = PR[GP1:90,2] + 8.377;
   1:L PR[91] R[100]mm/sec CNT100;
   1:  PR[GP1:91,1] = PR[GP1:90,1] + 5.462;
   1:  PR[GP1:91,2] = PR[GP1:90,2] + 7.189;
   1:L PR[91] R[100]mm/sec CNT100;
   1:  PR[GP1:91,1] = PR[GP1:90,1] + 6.729;
   1:  PR[GP1:91,2] = PR[GP1:90,2] + 7.060;
   1:L PR[91] R[100]mm/sec CNT100;
   1:  PR[GP1:91,1] = PR[GP1:90,1] + 4.245;
   1:  PR[GP1:91,2] = PR[GP1:90,2] + 4.798;
   1:L PR[91] R[100]mm/sec CNT100;
   1:  PR[GP1:91,1] = PR[GP1:90,1] + 4.084;
   1:  PR[GP1:91,2] = PR[GP1:90,2] + 4.555;
   1:L PR[91] R[100]mm/sec CNT100;
   1:  PR[GP1:91,1] = PR[GP1:90,1] + 3.762;
   1:  PR[GP1:91,2] = PR[GP1:90,2] + 4.136;
   1:L PR[91] R[100]mm/sec CNT100;
   1:  PR[GP1:91,1] = PR[GP1:90,1] + 2.797;
   1:  PR[GP1:91,2] = PR[GP1:90,2] + 3.488;
   1:L PR[91] R[100]mm/sec CNT100;
   1:  PR[GP1:91,1] = PR[GP1:90,1] + 1.763;
   1:  PR[GP1:91,2] = PR[GP1:90,2] + 3.278;
   1:L PR[91] R[100]mm/sec CNT100;
   1:  PR[GP1:91,1] = PR[GP1:90,1] + -1.639;
   1:L PR[91] R[100]mm/sec CNT100;
   1:  PR[91] = PR[90];
   1:  PR[GP1:91,1] = PR[GP1:90,1] + -2.644;
   1:  PR[GP1:91,2] = PR[GP1:90,2] + 3.782;
   1:  PR[GP1:91,3] = PR[GP1:90,3] + 11.285;
   1:L PR[91] R[100]mm/sec CNT100;
   1:  PR[GP1:91,1] = PR[GP1:90,1] + -3.633;
   1:  PR[GP1:91,2] = PR[GP1:90,2] + 4.451;
   1:L PR[91] R[100]mm/sec CNT100;
   1:  PR[GP1:91,1] = PR[GP1:90,1] + -4.037;
   1:  PR[GP1:91,2] = PR[GP1:90,2] + 5.032;
   1:L PR[91] R[100]mm/sec CNT100;
   1:  PR[GP1:91,1] = PR[GP1:90,1] + -4.381;
   1:  PR[GP1:91,2] = PR[GP1:90,2] + 5.447;
   1:L PR[91] R[100]mm/sec CNT100;
   1:  PR[GP1:91,1] = PR[GP1:90,1] + -5.466;
   1:  PR[GP1:91,2] = PR[GP1:90,2] + 7.901;
   1:L PR[91] R[100]mm/sec CNT100;
   1:  PR[GP1:91,1] = PR[GP1:90,1] + -6.628;
   1:  PR[GP1:91,2] = PR[GP1:90,2] + 10.030;
   1:L PR[91] R[100]mm/sec CNT100;
   1:  PR[GP1:91,1] = PR[GP1:90,1] + -8.323;
   1:  PR[GP1:91,2] = PR[GP1:90,2] + 12.135;
   1:L PR[91] R[100]mm/sec CNT100;
   1:  PR[GP1:91,1] = PR[GP1:90,1] + -9.743;
   1:  PR[GP1:91,2] = PR[GP1:90,2] + 13.646;
   1:L PR[91] R[100]mm/sec CNT100;
   1:  PR[GP1:91,1] = PR[GP1:90,1] + -12.290;
   1:  PR[GP1:91,2] = PR[GP1:90,2] + 15.509;
   1:L PR[91] R[100]mm/sec CNT100;
   1:  PR[GP1:91,1] = PR[GP1:90,1] + -13.679;
   1:  PR[GP1:91,2] = PR[GP1:90,2] + 16.387;
   1:L PR[91] R[100]mm/sec CNT100;
   1:  PR[GP1:91,1] = PR[GP1:90,1] + -17.081;
   1:  PR[GP1:91,2] = PR[GP1:90,2] + 17.718;
   1:L PR[91] R[100]mm/sec CNT100;
   1:  PR[GP1:91,1] = PR[GP1:90,1] + -18.201;
   1:  PR[GP1:91,2] = PR[GP1:90,2] + 18.082;
   1:L PR[91] R[100]mm/sec CNT100;
   1:  PR[GP1:91,1] = PR[GP1:90,1] + -22.311;
   1:  PR[GP1:91,2] = PR[GP1:90,2] + 18.557;
   1:L PR[91] R[100]mm/sec CNT100;
   1:  PR[GP1:91,1] = PR[GP1:90,1] + -23.034;
   1:  PR[GP1:91,2] = PR[GP1:90,2] + 18.604;
   1:L PR[91] R[100]mm/sec CNT100;
   1:  PR[GP1:91,1] = PR[GP1:90,1] + -27.555;
   1:  PR[GP1:91,2] = PR[GP1:90,2] + 17.956;
   1:L PR[91] R[100]mm/sec CNT100;
   1:  PR[GP1:91,1] = PR[GP1:90,1] + -27.868;
   1:  PR[GP1:91,2] = PR[GP1:90,2] + 17.898;
   1:L PR[91] R[100]mm/sec CNT100;
   1:  PR[GP1:91,1] = PR[GP1:90,1] + -32.403;
   1:  PR[GP1:91,2] = PR[GP1:90,2] + 15.975;
   1:L PR[91] R[100]mm/sec CNT100;
   1:  PR[GP1:91,1] = PR[GP1:90,1] + -36.273;
   1:  PR[GP1:91,2] = PR[GP1:90,2] + 12.982;
   1:L PR[91] R[100]mm/sec CNT100;
   1:  PR[GP1:91,1] = PR[GP1:90,1] + -39.253;
   1:  PR[GP1:91,2] = PR[GP1:90,2] + 9.082;
   1:L PR[91] R[100]mm/sec CNT100;
   1:  PR[GP1:91,1] = PR[GP1:90,1] + -39.260;
   1:  PR[GP1:91,2] = PR[GP1:90,2] + 9.064;
   1:L PR[91] R[100]mm/sec CNT100;
   1:  PR[GP1:91,1] = PR[GP1:90,1] + -41.123;
   1:  PR[GP1:91,2] = PR[GP1:90,2] + 4.556;
   1:L PR[91] R[100]mm/sec CNT100;
   1:  PR[GP1:91,1] = PR[GP1:90,1] + -41.130;
   1:  PR[GP1:91,2] = PR[GP1:90,2] + 4.529;
   1:L PR[91] R[100]mm/sec CNT100;
   1:  PR[GP1:91,1] = PR[GP1:90,1] + -41.752;
   1:  PR[GP1:91,2] = PR[GP1:90,2] + -0.345;
   1:L PR[91] R[100]mm/sec CNT100;
   1:  PR[GP1:91,1] = PR[GP1:90,1] + -41.741;
   1:  PR[GP1:91,2] = PR[GP1:90,2] + -0.476;
   1:L PR[91] R[100]mm/sec CNT100;
   1:  PR[GP1:91,1] = PR[GP1:90,1] + -41.130;
   1:  PR[GP1:91,2] = PR[GP1:90,2] + -5.151;
   1:L PR[91] R[100]mm/sec CNT100;
   1:  PR[GP1:91,1] = PR[GP1:90,1] + -41.123;
   1:  PR[GP1:91,2] = PR[GP1:90,2] + -5.180;
   1:L PR[91] R[100]mm/sec CNT100;
   1:  PR[GP1:91,1] = PR[GP1:90,1] + -39.247;
   1:  PR[GP1:91,2] = PR[GP1:90,2] + -9.713;
   1:L PR[91] R[100]mm/sec CNT100;
   1:  PR[GP1:91,1] = PR[GP1:90,1] + -36.306;
   1:  PR[GP1:91,2] = PR[GP1:90,2] + -13.570;
   1:L PR[91] R[100]mm/sec CNT100;
   1:  PR[GP1:91,1] = PR[GP1:90,1] + -32.402;
   1:  PR[GP1:91,2] = PR[GP1:90,2] + -16.600;
   1:L PR[91] R[100]mm/sec CNT100;
   1:  PR[GP1:91,1] = PR[GP1:90,1] + -27.869;
   1:  PR[GP1:91,2] = PR[GP1:90,2] + -18.522;
   1:L PR[91] R[100]mm/sec CNT100;
   1:  PR[GP1:91,1] = PR[GP1:90,1] + -27.556;
   1:  PR[GP1:91,2] = PR[GP1:90,2] + -18.580;
   1:L PR[91] R[100]mm/sec CNT100;
   1:  PR[GP1:91,1] = PR[GP1:90,1] + -23.035;
   1:  PR[GP1:91,2] = PR[GP1:90,2] + -19.228;
   1:L PR[91] R[100]mm/sec CNT100;
   1:  PR[GP1:91,1] = PR[GP1:90,1] + -22.311;
   1:  PR[GP1:91,2] = PR[GP1:90,2] + -19.181;
   1:L PR[91] R[100]mm/sec CNT100;
   1:  PR[GP1:91,1] = PR[GP1:90,1] + -18.202;
   1:  PR[GP1:91,2] = PR[GP1:90,2] + -18.706;
   1:L PR[91] R[100]mm/sec CNT100;
   1:  PR[GP1:91,1] = PR[GP1:90,1] + -17.081;
   1:  PR[GP1:91,2] = PR[GP1:90,2] + -18.342;
   1:L PR[91] R[100]mm/sec CNT100;
   1:  PR[GP1:91,1] = PR[GP1:90,1] + -13.679;
   1:  PR[GP1:91,2] = PR[GP1:90,2] + -17.011;
   1:L PR[91] R[100]mm/sec CNT100;
   1:  PR[GP1:91,1] = PR[GP1:90,1] + -12.290;
   1:  PR[GP1:91,2] = PR[GP1:90,2] + -16.133;
   1:L PR[91] R[100]mm/sec CNT100;
   1:  PR[GP1:91,1] = PR[GP1:90,1] + -9.743;
   1:  PR[GP1:91,2] = PR[GP1:90,2] + -14.270;
   1:L PR[91] R[100]mm/sec CNT100;
   1:  PR[GP1:91,1] = PR[GP1:90,1] + -8.324;
   1:  PR[GP1:91,2] = PR[GP1:90,2] + -12.759;
   1:L PR[91] R[100]mm/sec CNT100;
   1:  PR[GP1:91,1] = PR[GP1:90,1] + -6.627;
   1:  PR[GP1:91,2] = PR[GP1:90,2] + -10.654;
   1:L PR[91] R[100]mm/sec CNT100;
   1:  PR[GP1:91,1] = PR[GP1:90,1] + -5.467;
   1:  PR[GP1:91,2] = PR[GP1:90,2] + -8.528;
   1:L PR[91] R[100]mm/sec CNT100;
   1:  PR[GP1:91,1] = PR[GP1:90,1] + -4.362;
   1:  PR[GP1:91,2] = PR[GP1:90,2] + -6.027;
   1:L PR[91] R[100]mm/sec CNT100;
   1:  PR[GP1:91,1] = PR[GP1:90,1] + -4.108;
   1:  PR[GP1:91,2] = PR[GP1:90,2] + -5.758;
   1:L PR[91] R[100]mm/sec CNT100;
   1:  PR[GP1:91,1] = PR[GP1:90,1] + -3.633;
   1:  PR[GP1:91,2] = PR[GP1:90,2] + -5.075;
   1:L PR[91] R[100]mm/sec CNT100;
   1:  PR[GP1:91,1] = PR[GP1:90,1] + -2.642;
   1:  PR[GP1:91,2] = PR[GP1:90,2] + -4.405;
   1:L PR[91] R[100]mm/sec CNT100;
   1:  PR[GP1:91,1] = PR[GP1:90,1] + -1.620;
   1:  PR[GP1:91,2] = PR[GP1:90,2] + -4.190;
   1:L PR[91] R[100]mm/sec CNT100;
   1:  PR[GP1:91,1] = PR[GP1:90,1] + 1.763;
   1:L PR[91] R[100]mm/sec CNT100;
   1:  PR[GP1:91,1] = PR[GP1:90,1] + 2.793;
   1:  PR[GP1:91,2] = PR[GP1:90,2] + -4.403;
   1:L PR[91] R[100]mm/sec CNT100;
   1:  PR[GP1:91,1] = PR[GP1:90,1] + 3.787;
   1:  PR[GP1:91,2] = PR[GP1:90,2] + -5.073;
   1:L PR[91] R[100]mm/sec CNT100;
   1:  PR[GP1:91,1] = PR[GP1:90,1] + 4.266;
   1:  PR[GP1:91,2] = PR[GP1:90,2] + -5.763;
   1:L PR[91] R[100]mm/sec CNT100;
   1:  PR[GP1:91,1] = PR[GP1:90,1] + 4.516;
   1:  PR[GP1:91,2] = PR[GP1:90,2] + -6.034;
   1:L PR[91] R[100]mm/sec CNT100;
   1:  PR[GP1:91,1] = PR[GP1:90,1] + 5.617;
   1:  PR[GP1:91,2] = PR[GP1:90,2] + -8.514;
   1:L PR[91] R[100]mm/sec CNT100;
   1:  PR[GP1:91,1] = PR[GP1:90,1] + 6.782;
   1:  PR[GP1:91,2] = PR[GP1:90,2] + -10.647;
   1:L PR[91] R[100]mm/sec CNT100;
   1:  PR[GP1:91,1] = PR[GP1:90,1] + 8.479;
   1:  PR[GP1:91,2] = PR[GP1:90,2] + -12.755;
   1:L PR[91] R[100]mm/sec CNT100;
   1:  PR[GP1:91,1] = PR[GP1:90,1] + 9.899;
   1:  PR[GP1:91,2] = PR[GP1:90,2] + -14.269;
   1:L PR[91] R[100]mm/sec CNT100;
   1:  PR[GP1:91,1] = PR[GP1:90,1] + 12.444;
   1:  PR[GP1:91,2] = PR[GP1:90,2] + -16.132;
   1:L PR[91] R[100]mm/sec CNT100;
   1:  PR[GP1:91,1] = PR[GP1:90,1] + 13.833;
   1:  PR[GP1:91,2] = PR[GP1:90,2] + -17.010;
   1:L PR[91] R[100]mm/sec CNT100;
   1:  PR[GP1:91,1] = PR[GP1:90,1] + 17.235;
   1:  PR[GP1:91,2] = PR[GP1:90,2] + -18.341;
   1:L PR[91] R[100]mm/sec CNT100;
   1:  PR[GP1:91,1] = PR[GP1:90,1] + 18.357;
   1:  PR[GP1:91,2] = PR[GP1:90,2] + -18.705;
   1:L PR[91] R[100]mm/sec CNT100;
   1:  PR[GP1:91,1] = PR[GP1:90,1] + 22.466;
   1:  PR[GP1:91,2] = PR[GP1:90,2] + -19.181;
   1:L PR[91] R[100]mm/sec CNT100;
   1:  PR[GP1:91,1] = PR[GP1:90,1] + 23.190;
   1:  PR[GP1:91,2] = PR[GP1:90,2] + -19.228;
   1:L PR[91] R[100]mm/sec CNT100;
   1:  PR[GP1:91,1] = PR[GP1:90,1] + 27.711;
   1:  PR[GP1:91,2] = PR[GP1:90,2] + -18.580;
   1:L PR[91] R[100]mm/sec CNT100;
   1:  PR[GP1:91,1] = PR[GP1:90,1] + 28.024;
   1:  PR[GP1:91,2] = PR[GP1:90,2] + -18.522;
   1:L PR[91] R[100]mm/sec CNT100;
   1:  PR[GP1:91,1] = PR[GP1:90,1] + 32.559;
   1:  PR[GP1:91,2] = PR[GP1:90,2] + -16.600;
   1:L PR[91] R[100]mm/sec CNT100;
   1:  PR[GP1:91,1] = PR[GP1:90,1] + 36.429;
   1:  PR[GP1:91,2] = PR[GP1:90,2] + -13.606;
   1:L PR[91] R[100]mm/sec CNT100;
   1:  PR[GP1:91,1] = PR[GP1:90,1] + 39.404;
   1:  PR[GP1:91,2] = PR[GP1:90,2] + -9.712;
   1:L PR[91] R[100]mm/sec CNT100;
   1:  PR[GP1:91,1] = PR[GP1:90,1] + 41.280;
   1:  PR[GP1:91,2] = PR[GP1:90,2] + -5.183;
   1:L PR[91] R[100]mm/sec CNT100;
   1:  PR[GP1:91,1] = PR[GP1:90,1] + 41.287;
   1:  PR[GP1:91,2] = PR[GP1:90,2] + -5.156;
   1:L PR[91] R[100]mm/sec CNT100;
   1:  PR[GP1:91,1] = PR[GP1:90,1] + 41.909;
   1:  PR[GP1:91,2] = PR[GP1:90,2] + -0.279;
   1:L PR[91] R[100]mm/sec CNT100;
   1:  PR[GP1:91,1] = PR[GP1:90,1] + 41.898;
   1:  PR[GP1:91,2] = PR[GP1:90,2] + -0.148;
   1:L PR[91] R[100]mm/sec CNT100;
   1:  PR[GP1:91,1] = PR[GP1:90,1] + 41.287;
   1:  PR[GP1:91,2] = PR[GP1:90,2] + 4.531;
   1:L PR[91] R[100]mm/sec CNT100;
   1:  PR[GP1:91,1] = PR[GP1:90,1] + 41.280;
   1:  PR[GP1:91,2] = PR[GP1:90,2] + 4.560;
   1:L PR[91] R[100]mm/sec CNT100;
   1:  PR[GP1:91,1] = PR[GP1:90,1] + 39.403;
   1:  PR[GP1:91,2] = PR[GP1:90,2] + 9.090;
   1:L PR[91] R[100]mm/sec CNT100;
   1:  PR[GP1:91,1] = PR[GP1:90,1] + 36.427;
   1:  PR[GP1:91,2] = PR[GP1:90,2] + 12.985;
   1:L PR[91] R[100]mm/sec CNT100;
   1:  PR[GP1:91,1] = PR[GP1:90,1] + 32.556;
   1:  PR[GP1:91,2] = PR[GP1:90,2] + 15.978;
   1:L PR[91] R[100]mm/sec CNT100;
   1:  PR[GP1:91,1] = PR[GP1:90,1] + 28.019;
   1:  PR[GP1:91,2] = PR[GP1:90,2] + 17.900;
   1:L PR[91] R[100]mm/sec CNT100;
   1:  PR[GP1:91,1] = PR[GP1:90,1] + 27.706;
   1:  PR[GP1:91,2] = PR[GP1:90,2] + 17.958;
   1:L PR[91] R[100]mm/sec CNT100;
   1:  PR[GP1:91,1] = PR[GP1:90,1] + 23.185;
   1:  PR[GP1:91,2] = PR[GP1:90,2] + 18.604;
   1:L PR[91] R[100]mm/sec CNT100;
   1:  PR[GP1:91,1] = PR[GP1:90,1] + 22.461;
   1:  PR[GP1:91,2] = PR[GP1:90,2] + 18.557;
   1:L PR[91] R[100]mm/sec CNT100;
   1:  PR[GP1:91,1] = PR[GP1:90,1] + 18.352;
   1:  PR[GP1:91,2] = PR[GP1:90,2] + 18.080;
   1:L PR[91] R[100]mm/sec CNT100;
   1:  PR[GP1:91,1] = PR[GP1:90,1] + 17.231;
   1:  PR[GP1:91,2] = PR[GP1:90,2] + 17.716;
   1:L PR[91] R[100]mm/sec CNT100;
   1:  PR[GP1:91,1] = PR[GP1:90,1] + 13.829;
   1:  PR[GP1:91,2] = PR[GP1:90,2] + 16.384;
   1:L PR[91] R[100]mm/sec CNT100;
   1:  PR[GP1:91,1] = PR[GP1:90,1] + 12.441;
   1:  PR[GP1:91,2] = PR[GP1:90,2] + 15.506;
   1:L PR[91] R[100]mm/sec CNT100;
   1:  PR[GP1:91,1] = PR[GP1:90,1] + 9.896;
   1:  PR[GP1:91,2] = PR[GP1:90,2] + 13.643;
   1:L PR[91] R[100]mm/sec CNT100;
   1:  PR[GP1:91,1] = PR[GP1:90,1] + 8.477;
   1:  PR[GP1:91,2] = PR[GP1:90,2] + 12.129;
   1:L PR[91] R[100]mm/sec CNT100;
   1:  PR[GP1:91,1] = PR[GP1:90,1] + 6.781;
   1:  PR[GP1:91,2] = PR[GP1:90,2] + 10.020;
   1:L PR[91] R[100]mm/sec CNT100;
   1:  PR[GP1:91,1] = PR[GP1:90,1] + 5.623;
   1:  PR[GP1:91,2] = PR[GP1:90,2] + 7.906;
   1:L PR[91] R[100]mm/sec CNT100;
   1:  PR[GP1:91,1] = PR[GP1:90,1] + 5.419;
   1:  PR[GP1:91,2] = PR[GP1:90,2] + 7.443;
   1:L PR[91] R[100]mm/sec CNT100;
   1:  PR[GP1:91,1] = PR[GP1:90,1] + 6.860;
   1:  PR[GP1:91,2] = PR[GP1:90,2] + 7.296;
   1:L PR[91] R[100]mm/sec CNT100;
   1:  PR[GP1:91,1] = PR[GP1:90,1] + 4.215;
   1:  PR[GP1:91,2] = PR[GP1:90,2] + 5.065;
   1:L PR[91] R[100]mm/sec CNT100;
   1:  PR[GP1:91,1] = PR[GP1:90,1] + 3.789;
   1:  PR[GP1:91,2] = PR[GP1:90,2] + 4.452;
   1:L PR[91] R[100]mm/sec CNT100;
   1:  PR[GP1:91,1] = PR[GP1:90,1] + 2.794;
   1:  PR[GP1:91,2] = PR[GP1:90,2] + 3.778;
   1:L PR[91] R[100]mm/sec CNT100;
   1:  PR[GP1:91,1] = PR[GP1:90,1] + 1.754;
   1:  PR[GP1:91,2] = PR[GP1:90,2] + 3.566;
   1:L PR[91] R[100]mm/sec CNT100;
   1:  PR[GP1:91,1] = PR[GP1:90,1] + -1.635;
   1:L PR[91] R[100]mm/sec CNT100;
   1:  PR[91] = PR[90];
   1:  PR[GP1:91,1] = PR[GP1:90,1] + -2.643;
   1:  PR[GP1:91,2] = PR[GP1:90,2] + 4.074;
   1:  PR[GP1:91,3] = PR[GP1:90,3] + 11.895;
   1:L PR[91] R[100]mm/sec CNT100;
   1:  PR[GP1:91,1] = PR[GP1:90,1] + -3.634;
   1:  PR[GP1:91,2] = PR[GP1:90,2] + 4.749;
   1:L PR[91] R[100]mm/sec CNT100;
   1:  PR[GP1:91,1] = PR[GP1:90,1] + -4.032;
   1:  PR[GP1:91,2] = PR[GP1:90,2] + 5.326;
   1:L PR[91] R[100]mm/sec CNT100;
   1:  PR[GP1:91,1] = PR[GP1:90,1] + -4.343;
   1:  PR[GP1:91,2] = PR[GP1:90,2] + 5.702;
   1:L PR[91] R[100]mm/sec CNT100;
   1:  PR[GP1:91,1] = PR[GP1:90,1] + -5.101;
   1:  PR[GP1:91,2] = PR[GP1:90,2] + 7.425;
   1:L PR[91] R[100]mm/sec CNT100;
   1:  PR[GP1:91,1] = PR[GP1:90,1] + -6.633;
   1:  PR[GP1:91,2] = PR[GP1:90,2] + 10.232;
   1:L PR[91] R[100]mm/sec CNT100;
   1:  PR[GP1:91,1] = PR[GP1:90,1] + -7.844;
   1:  PR[GP1:91,2] = PR[GP1:90,2] + 11.734;
   1:L PR[91] R[100]mm/sec CNT100;
   1:  PR[GP1:91,1] = PR[GP1:90,1] + -9.776;
   1:  PR[GP1:91,2] = PR[GP1:90,2] + 13.791;
   1:L PR[91] R[100]mm/sec CNT100;
   1:  PR[GP1:91,1] = PR[GP1:90,1] + -11.725;
   1:  PR[GP1:91,2] = PR[GP1:90,2] + 15.216;
   1:L PR[91] R[100]mm/sec CNT100;
   1:  PR[GP1:91,1] = PR[GP1:90,1] + -13.720;
   1:  PR[GP1:91,2] = PR[GP1:90,2] + 16.478;
   1:L PR[91] R[100]mm/sec CNT100;
   1:  PR[GP1:91,1] = PR[GP1:90,1] + -16.469;
   1:  PR[GP1:91,2] = PR[GP1:90,2] + 17.553;
   1:L PR[91] R[100]mm/sec CNT100;
   1:  PR[GP1:91,1] = PR[GP1:90,1] + -18.237;
   1:  PR[GP1:91,2] = PR[GP1:90,2] + 18.128;
   1:L PR[91] R[100]mm/sec CNT100;
   1:  PR[GP1:91,1] = PR[GP1:90,1] + -21.692;
   1:  PR[GP1:91,2] = PR[GP1:90,2] + 18.527;
   1:L PR[91] R[100]mm/sec CNT100;
   1:  PR[GP1:91,1] = PR[GP1:90,1] + -23.055;
   1:  PR[GP1:91,2] = PR[GP1:90,2] + 18.616;
   1:L PR[91] R[100]mm/sec CNT100;
   1:  PR[GP1:91,1] = PR[GP1:90,1] + -26.965;
   1:  PR[GP1:91,2] = PR[GP1:90,2] + 18.056;
   1:L PR[91] R[100]mm/sec CNT100;
   1:  PR[GP1:91,1] = PR[GP1:90,1] + -27.870;
   1:  PR[GP1:91,2] = PR[GP1:90,2] + 17.888;
   1:L PR[91] R[100]mm/sec CNT100;
   1:  PR[GP1:91,1] = PR[GP1:90,1] + -31.868;
   1:  PR[GP1:91,2] = PR[GP1:90,2] + 16.198;
   1:L PR[91] R[100]mm/sec CNT100;
   1:  PR[GP1:91,1] = PR[GP1:90,1] + -32.365;
   1:  PR[GP1:91,2] = PR[GP1:90,2] + 15.968;
   1:L PR[91] R[100]mm/sec CNT100;
   1:  PR[GP1:91,1] = PR[GP1:90,1] + -36.035;
   1:  PR[GP1:91,2] = PR[GP1:90,2] + 13.131;
   1:L PR[91] R[100]mm/sec CNT100;
   1:  PR[GP1:91,1] = PR[GP1:90,1] + -36.234;
   1:  PR[GP1:91,2] = PR[GP1:90,2] + 12.968;
   1:L PR[91] R[100]mm/sec CNT100;
   1:  PR[GP1:91,1] = PR[GP1:90,1] + -39.215;
   1:  PR[GP1:91,2] = PR[GP1:90,2] + 9.060;
   1:L PR[91] R[100]mm/sec CNT100;
   1:  PR[GP1:91,1] = PR[GP1:90,1] + -41.085;
   1:  PR[GP1:91,2] = PR[GP1:90,2] + 4.544;
   1:L PR[91] R[100]mm/sec CNT100;
   1:  PR[GP1:91,1] = PR[GP1:90,1] + -41.726;
   1:  PR[GP1:91,2] = PR[GP1:90,2] + -0.312;
   1:L PR[91] R[100]mm/sec CNT100;
   1:  PR[GP1:91,1] = PR[GP1:90,1] + -41.085;
   1:  PR[GP1:91,2] = PR[GP1:90,2] + -5.168;
   1:L PR[91] R[100]mm/sec CNT100;
   1:  PR[GP1:91,1] = PR[GP1:90,1] + -39.215;
   1:  PR[GP1:91,2] = PR[GP1:90,2] + -9.684;
   1:L PR[91] R[100]mm/sec CNT100;
   1:  PR[GP1:91,1] = PR[GP1:90,1] + -36.234;
   1:  PR[GP1:91,2] = PR[GP1:90,2] + -13.592;
   1:L PR[91] R[100]mm/sec CNT100;
   1:  PR[GP1:91,1] = PR[GP1:90,1] + -36.034;
   1:  PR[GP1:91,2] = PR[GP1:90,2] + -13.755;
   1:L PR[91] R[100]mm/sec CNT100;
   1:  PR[GP1:91,1] = PR[GP1:90,1] + -32.365;
   1:  PR[GP1:91,2] = PR[GP1:90,2] + -16.591;
   1:L PR[91] R[100]mm/sec CNT100;
   1:  PR[GP1:91,1] = PR[GP1:90,1] + -31.868;
   1:  PR[GP1:91,2] = PR[GP1:90,2] + -16.821;
   1:L PR[91] R[100]mm/sec CNT100;
   1:  PR[GP1:91,1] = PR[GP1:90,1] + -27.870;
   1:  PR[GP1:91,2] = PR[GP1:90,2] + -18.512;
   1:L PR[91] R[100]mm/sec CNT100;
   1:  PR[GP1:91,1] = PR[GP1:90,1] + -26.965;
   1:  PR[GP1:91,2] = PR[GP1:90,2] + -18.680;
   1:L PR[91] R[100]mm/sec CNT100;
   1:  PR[GP1:91,1] = PR[GP1:90,1] + -23.055;
   1:  PR[GP1:91,2] = PR[GP1:90,2] + -19.240;
   1:L PR[91] R[100]mm/sec CNT100;
   1:  PR[GP1:91,1] = PR[GP1:90,1] + -21.692;
   1:  PR[GP1:91,2] = PR[GP1:90,2] + -19.151;
   1:L PR[91] R[100]mm/sec CNT100;
   1:  PR[GP1:91,1] = PR[GP1:90,1] + -18.238;
   1:  PR[GP1:91,2] = PR[GP1:90,2] + -18.752;
   1:L PR[91] R[100]mm/sec CNT100;
   1:  PR[GP1:91,1] = PR[GP1:90,1] + -16.469;
   1:  PR[GP1:91,2] = PR[GP1:90,2] + -18.177;
   1:L PR[91] R[100]mm/sec CNT100;
   1:  PR[GP1:91,1] = PR[GP1:90,1] + -13.720;
   1:  PR[GP1:91,2] = PR[GP1:90,2] + -17.102;
   1:L PR[91] R[100]mm/sec CNT100;
   1:  PR[GP1:91,1] = PR[GP1:90,1] + -11.725;
   1:  PR[GP1:91,2] = PR[GP1:90,2] + -15.840;
   1:L PR[91] R[100]mm/sec CNT100;
   1:  PR[GP1:91,1] = PR[GP1:90,1] + -9.776;
   1:  PR[GP1:91,2] = PR[GP1:90,2] + -14.415;
   1:L PR[91] R[100]mm/sec CNT100;
   1:  PR[GP1:91,1] = PR[GP1:90,1] + -7.843;
   1:  PR[GP1:91,2] = PR[GP1:90,2] + -12.358;
   1:L PR[91] R[100]mm/sec CNT100;
   1:  PR[GP1:91,1] = PR[GP1:90,1] + -6.633;
   1:  PR[GP1:91,2] = PR[GP1:90,2] + -10.855;
   1:L PR[91] R[100]mm/sec CNT100;
   1:  PR[GP1:91,1] = PR[GP1:90,1] + -5.103;
   1:  PR[GP1:91,2] = PR[GP1:90,2] + -8.052;
   1:L PR[91] R[100]mm/sec CNT100;
   1:  PR[GP1:91,1] = PR[GP1:90,1] + -4.315;
   1:  PR[GP1:91,2] = PR[GP1:90,2] + -6.269;
   1:L PR[91] R[100]mm/sec CNT100;
   1:  PR[GP1:91,1] = PR[GP1:90,1] + -4.099;
   1:  PR[GP1:91,2] = PR[GP1:90,2] + -6.048;
   1:L PR[91] R[100]mm/sec CNT100;
   1:  PR[GP1:91,1] = PR[GP1:90,1] + -3.633;
   1:  PR[GP1:91,2] = PR[GP1:90,2] + -5.372;
   1:L PR[91] R[100]mm/sec CNT100;
   1:  PR[GP1:91,1] = PR[GP1:90,1] + -2.639;
   1:  PR[GP1:91,2] = PR[GP1:90,2] + -4.696;
   1:L PR[91] R[100]mm/sec CNT100;
   1:  PR[GP1:91,1] = PR[GP1:90,1] + -1.614;
   1:  PR[GP1:91,2] = PR[GP1:90,2] + -4.479;
   1:L PR[91] R[100]mm/sec CNT100;
   1:  PR[GP1:91,1] = PR[GP1:90,1] + 1.755;
   1:L PR[91] R[100]mm/sec CNT100;
   1:  PR[GP1:91,1] = PR[GP1:90,1] + 2.790;
   1:  PR[GP1:91,2] = PR[GP1:90,2] + -4.694;
   1:L PR[91] R[100]mm/sec CNT100;
   1:  PR[GP1:91,1] = PR[GP1:90,1] + 3.787;
   1:  PR[GP1:91,2] = PR[GP1:90,2] + -5.371;
   1:L PR[91] R[100]mm/sec CNT100;
   1:  PR[GP1:91,1] = PR[GP1:90,1] + 4.256;
   1:  PR[GP1:91,2] = PR[GP1:90,2] + -6.052;
   1:L PR[91] R[100]mm/sec CNT100;
   1:  PR[GP1:91,1] = PR[GP1:90,1] + 4.469;
   1:  PR[GP1:91,2] = PR[GP1:90,2] + -6.274;
   1:L PR[91] R[100]mm/sec CNT100;
   1:  PR[GP1:91,1] = PR[GP1:90,1] + 5.251;
   1:  PR[GP1:91,2] = PR[GP1:90,2] + -8.036;
   1:L PR[91] R[100]mm/sec CNT100;
   1:  PR[GP1:91,1] = PR[GP1:90,1] + 6.787;
   1:  PR[GP1:91,2] = PR[GP1:90,2] + -10.848;
   1:L PR[91] R[100]mm/sec CNT100;
   1:  PR[GP1:91,1] = PR[GP1:90,1] + 7.998;
   1:  PR[GP1:91,2] = PR[GP1:90,2] + -12.352;
   1:L PR[91] R[100]mm/sec CNT100;
   1:  PR[GP1:91,1] = PR[GP1:90,1] + 9.931;
   1:  PR[GP1:91,2] = PR[GP1:90,2] + -14.414;
   1:L PR[91] R[100]mm/sec CNT100;
   1:  PR[GP1:91,1] = PR[GP1:90,1] + 11.879;
   1:  PR[GP1:91,2] = PR[GP1:90,2] + -15.839;
   1:L PR[91] R[100]mm/sec CNT100;
   1:  PR[GP1:91,1] = PR[GP1:90,1] + 13.874;
   1:  PR[GP1:91,2] = PR[GP1:90,2] + -17.100;
   1:L PR[91] R[100]mm/sec CNT100;
   1:  PR[GP1:91,1] = PR[GP1:90,1] + 16.623;
   1:  PR[GP1:91,2] = PR[GP1:90,2] + -18.176;
   1:L PR[91] R[100]mm/sec CNT100;
   1:  PR[GP1:91,1] = PR[GP1:90,1] + 18.392;
   1:  PR[GP1:91,2] = PR[GP1:90,2] + -18.751;
   1:L PR[91] R[100]mm/sec CNT100;
   1:  PR[GP1:91,1] = PR[GP1:90,1] + 21.846;
   1:  PR[GP1:91,2] = PR[GP1:90,2] + -19.151;
   1:L PR[91] R[100]mm/sec CNT100;
   1:  PR[GP1:91,1] = PR[GP1:90,1] + 23.210;
   1:  PR[GP1:91,2] = PR[GP1:90,2] + -19.240;
   1:L PR[91] R[100]mm/sec CNT100;
   1:  PR[GP1:91,1] = PR[GP1:90,1] + 27.120;
   1:  PR[GP1:91,2] = PR[GP1:90,2] + -18.680;
   1:L PR[91] R[100]mm/sec CNT100;
   1:  PR[GP1:91,1] = PR[GP1:90,1] + 28.026;
   1:  PR[GP1:91,2] = PR[GP1:90,2] + -18.512;
   1:L PR[91] R[100]mm/sec CNT100;
   1:  PR[GP1:91,1] = PR[GP1:90,1] + 32.024;
   1:  PR[GP1:91,2] = PR[GP1:90,2] + -16.822;
   1:L PR[91] R[100]mm/sec CNT100;
   1:  PR[GP1:91,1] = PR[GP1:90,1] + 32.521;
   1:  PR[GP1:91,2] = PR[GP1:90,2] + -16.592;
   1:L PR[91] R[100]mm/sec CNT100;
   1:  PR[GP1:91,1] = PR[GP1:90,1] + 36.190;
   1:  PR[GP1:91,2] = PR[GP1:90,2] + -13.756;
   1:L PR[91] R[100]mm/sec CNT100;
   1:  PR[GP1:91,1] = PR[GP1:90,1] + 36.390;
   1:  PR[GP1:91,2] = PR[GP1:90,2] + -13.593;
   1:L PR[91] R[100]mm/sec CNT100;
   1:  PR[GP1:91,1] = PR[GP1:90,1] + 39.372;
   1:  PR[GP1:91,2] = PR[GP1:90,2] + -9.682;
   1:L PR[91] R[100]mm/sec CNT100;
   1:  PR[GP1:91,1] = PR[GP1:90,1] + 41.242;
   1:  PR[GP1:91,2] = PR[GP1:90,2] + -5.172;
   1:L PR[91] R[100]mm/sec CNT100;
   1:  PR[GP1:91,1] = PR[GP1:90,1] + 41.720;
   1:  PR[GP1:91,2] = PR[GP1:90,2] + -1.566;
   1:L PR[91] R[100]mm/sec CNT100;
   1:  PR[GP1:91,1] = PR[GP1:90,1] + 41.883;
   1:  PR[GP1:91,2] = PR[GP1:90,2] + -0.314;
   1:L PR[91] R[100]mm/sec CNT100;
   1:  PR[GP1:91,1] = PR[GP1:90,1] + 41.242;
   1:  PR[GP1:91,2] = PR[GP1:90,2] + 4.549;
   1:L PR[91] R[100]mm/sec CNT100;
   1:  PR[GP1:91,1] = PR[GP1:90,1] + 39.371;
   1:  PR[GP1:91,2] = PR[GP1:90,2] + 9.060;
   1:L PR[91] R[100]mm/sec CNT100;
   1:  PR[GP1:91,1] = PR[GP1:90,1] + 36.388;
   1:  PR[GP1:91,2] = PR[GP1:90,2] + 12.971;
   1:L PR[91] R[100]mm/sec CNT100;
   1:  PR[GP1:91,1] = PR[GP1:90,1] + 36.188;
   1:  PR[GP1:91,2] = PR[GP1:90,2] + 13.134;
   1:L PR[91] R[100]mm/sec CNT100;
   1:  PR[GP1:91,1] = PR[GP1:90,1] + 32.518;
   1:  PR[GP1:91,2] = PR[GP1:90,2] + 15.970;
   1:L PR[91] R[100]mm/sec CNT100;
   1:  PR[GP1:91,1] = PR[GP1:90,1] + 32.021;
   1:  PR[GP1:91,2] = PR[GP1:90,2] + 16.200;
   1:L PR[91] R[100]mm/sec CNT100;
   1:  PR[GP1:91,1] = PR[GP1:90,1] + 28.022;
   1:  PR[GP1:91,2] = PR[GP1:90,2] + 17.889;
   1:L PR[91] R[100]mm/sec CNT100;
   1:  PR[GP1:91,1] = PR[GP1:90,1] + 27.117;
   1:  PR[GP1:91,2] = PR[GP1:90,2] + 18.057;
   1:L PR[91] R[100]mm/sec CNT100;
   1:  PR[GP1:91,1] = PR[GP1:90,1] + 23.207;
   1:  PR[GP1:91,2] = PR[GP1:90,2] + 18.616;
   1:L PR[91] R[100]mm/sec CNT100;
   1:  PR[GP1:91,1] = PR[GP1:90,1] + 21.843;
   1:  PR[GP1:91,2] = PR[GP1:90,2] + 18.527;
   1:L PR[91] R[100]mm/sec CNT100;
   1:  PR[GP1:91,1] = PR[GP1:90,1] + 18.389;
   1:  PR[GP1:91,2] = PR[GP1:90,2] + 18.126;
   1:L PR[91] R[100]mm/sec CNT100;
   1:  PR[GP1:91,1] = PR[GP1:90,1] + 16.621;
   1:  PR[GP1:91,2] = PR[GP1:90,2] + 17.552;
   1:L PR[91] R[100]mm/sec CNT100;
   1:  PR[GP1:91,1] = PR[GP1:90,1] + 13.872;
   1:  PR[GP1:91,2] = PR[GP1:90,2] + 16.475;
   1:L PR[91] R[100]mm/sec CNT100;
   1:  PR[GP1:91,1] = PR[GP1:90,1] + 11.877;
   1:  PR[GP1:91,2] = PR[GP1:90,2] + 15.215;
   1:L PR[91] R[100]mm/sec CNT100;
   1:  PR[GP1:91,1] = PR[GP1:90,1] + 9.930;
   1:  PR[GP1:91,2] = PR[GP1:90,2] + 13.789;
   1:L PR[91] R[100]mm/sec CNT100;
   1:  PR[GP1:91,1] = PR[GP1:90,1] + 7.998;
   1:  PR[GP1:91,2] = PR[GP1:90,2] + 11.729;
   1:L PR[91] R[100]mm/sec CNT100;
   1:  PR[GP1:91,1] = PR[GP1:90,1] + 6.787;
   1:  PR[GP1:91,2] = PR[GP1:90,2] + 10.223;
   1:L PR[91] R[100]mm/sec CNT100;
   1:  PR[GP1:91,1] = PR[GP1:90,1] + 5.403;
   1:  PR[GP1:91,2] = PR[GP1:90,2] + 7.695;
   1:L PR[91] R[100]mm/sec CNT100;
   1:  PR[GP1:91,1] = PR[GP1:90,1] + 6.846;
   1:  PR[GP1:91,2] = PR[GP1:90,2] + 7.549;
   1:L PR[91] R[100]mm/sec CNT100;
   1:  PR[GP1:91,1] = PR[GP1:90,1] + 4.210;
   1:  PR[GP1:91,2] = PR[GP1:90,2] + 5.361;
   1:L PR[91] R[100]mm/sec CNT100;
   1:  PR[GP1:91,1] = PR[GP1:90,1] + 3.794;
   1:  PR[GP1:91,2] = PR[GP1:90,2] + 4.756;
   1:L PR[91] R[100]mm/sec CNT100;
   1:  PR[GP1:91,1] = PR[GP1:90,1] + 3.146;
   1:  PR[GP1:91,2] = PR[GP1:90,2] + 4.304;
   1:L PR[91] R[100]mm/sec CNT100;
   1:  PR[GP1:91,1] = PR[GP1:90,1] + 2.767;
   1:  PR[GP1:91,2] = PR[GP1:90,2] + 4.064;
   1:L PR[91] R[100]mm/sec CNT100;
   1:  PR[GP1:91,1] = PR[GP1:90,1] + 1.746;
   1:  PR[GP1:91,2] = PR[GP1:90,2] + 3.855;
   1:L PR[91] R[100]mm/sec CNT100;
   1:  PR[GP1:91,1] = PR[GP1:90,1] + -1.631;
   1:L PR[91] R[100]mm/sec CNT100;
   1:  PR[91] = PR[90];
   1:  PR[GP1:91,1] = PR[GP1:90,1] + -2.641;
   1:  PR[GP1:91,2] = PR[GP1:90,2] + 4.365;
   1:  PR[GP1:91,3] = PR[GP1:90,3] + 12.505;
   1:L PR[91] R[100]mm/sec CNT100;
   1:  PR[GP1:91,1] = PR[GP1:90,1] + -3.634;
   1:  PR[GP1:91,2] = PR[GP1:90,2] + 5.047;
   1:L PR[91] R[100]mm/sec CNT100;
   1:  PR[GP1:91,1] = PR[GP1:90,1] + -4.070;
   1:  PR[GP1:91,2] = PR[GP1:90,2] + 5.685;
   1:L PR[91] R[100]mm/sec CNT100;
   1:  PR[GP1:91,1] = PR[GP1:90,1] + -4.261;
   1:  PR[GP1:91,2] = PR[GP1:90,2] + 5.854;
   1:L PR[91] R[100]mm/sec CNT100;
   1:  PR[GP1:91,1] = PR[GP1:90,1] + -4.738;
   1:  PR[GP1:91,2] = PR[GP1:90,2] + 6.952;
   1:L PR[91] R[100]mm/sec CNT100;
   1:  PR[GP1:91,1] = PR[GP1:90,1] + -6.639;
   1:  PR[GP1:91,2] = PR[GP1:90,2] + 10.433;
   1:L PR[91] R[100]mm/sec CNT100;
   1:  PR[GP1:91,1] = PR[GP1:90,1] + -7.364;
   1:  PR[GP1:91,2] = PR[GP1:90,2] + 11.334;
   1:L PR[91] R[100]mm/sec CNT100;
   1:  PR[GP1:91,1] = PR[GP1:90,1] + -9.809;
   1:  PR[GP1:91,2] = PR[GP1:90,2] + 13.935;
   1:L PR[91] R[100]mm/sec CNT100;
   1:  PR[GP1:91,1] = PR[GP1:90,1] + -11.160;
   1:  PR[GP1:91,2] = PR[GP1:90,2] + 14.923;
   1:L PR[91] R[100]mm/sec CNT100;
   1:  PR[GP1:91,1] = PR[GP1:90,1] + -13.762;
   1:  PR[GP1:91,2] = PR[GP1:90,2] + 16.568;
   1:L PR[91] R[100]mm/sec CNT100;
   1:  PR[GP1:91,1] = PR[GP1:90,1] + -15.857;
   1:  PR[GP1:91,2] = PR[GP1:90,2] + 17.388;
   1:L PR[91] R[100]mm/sec CNT100;
   1:  PR[GP1:91,1] = PR[GP1:90,1] + -18.273;
   1:  PR[GP1:91,2] = PR[GP1:90,2] + 18.174;
   1:L PR[91] R[100]mm/sec CNT100;
   1:  PR[GP1:91,1] = PR[GP1:90,1] + -21.073;
   1:  PR[GP1:91,2] = PR[GP1:90,2] + 18.497;
   1:L PR[91] R[100]mm/sec CNT100;
   1:  PR[GP1:91,1] = PR[GP1:90,1] + -23.076;
   1:  PR[GP1:91,2] = PR[GP1:90,2] + 18.628;
   1:L PR[91] R[100]mm/sec CNT100;
   1:  PR[GP1:91,1] = PR[GP1:90,1] + -26.375;
   1:  PR[GP1:91,2] = PR[GP1:90,2] + 18.155;
   1:L PR[91] R[100]mm/sec CNT100;
   1:  PR[GP1:91,1] = PR[GP1:90,1] + -27.871;
   1:  PR[GP1:91,2] = PR[GP1:90,2] + 17.877;
   1:L PR[91] R[100]mm/sec CNT100;
   1:  PR[GP1:91,1] = PR[GP1:90,1] + -31.336;
   1:  PR[GP1:91,2] = PR[GP1:90,2] + 16.412;
   1:L PR[91] R[100]mm/sec CNT100;
   1:  PR[GP1:91,1] = PR[GP1:90,1] + -32.345;
   1:  PR[GP1:91,2] = PR[GP1:90,2] + 15.945;
   1:L PR[91] R[100]mm/sec CNT100;
   1:  PR[GP1:91,1] = PR[GP1:90,1] + -35.584;
   1:  PR[GP1:91,2] = PR[GP1:90,2] + 13.442;
   1:L PR[91] R[100]mm/sec CNT100;
   1:  PR[GP1:91,1] = PR[GP1:90,1] + -36.196;
   1:  PR[GP1:91,2] = PR[GP1:90,2] + 12.943;
   1:L PR[91] R[100]mm/sec CNT100;
   1:  PR[GP1:91,1] = PR[GP1:90,1] + -38.824;
   1:  PR[GP1:91,2] = PR[GP1:90,2] + 9.505;
   1:L PR[91] R[100]mm/sec CNT100;
   1:  PR[GP1:91,1] = PR[GP1:90,1] + -39.156;
   1:  PR[GP1:91,2] = PR[GP1:90,2] + 9.052;
   1:L PR[91] R[100]mm/sec CNT100;
   1:  PR[GP1:91,1] = PR[GP1:90,1] + -41.023;
   1:  PR[GP1:91,2] = PR[GP1:90,2] + 4.535;
   1:L PR[91] R[100]mm/sec CNT100;
   1:  PR[GP1:91,1] = PR[GP1:90,1] + -41.664;
   1:  PR[GP1:91,2] = PR[GP1:90,2] + -0.312;
   1:L PR[91] R[100]mm/sec CNT100;
   1:  PR[GP1:91,1] = PR[GP1:90,1] + -41.023;
   1:  PR[GP1:91,2] = PR[GP1:90,2] + -5.159;
   1:L PR[91] R[100]mm/sec CNT100;
   1:  PR[GP1:91,1] = PR[GP1:90,1] + -39.157;
   1:  PR[GP1:91,2] = PR[GP1:90,2] + -9.675;
   1:L PR[91] R[100]mm/sec CNT100;
   1:  PR[GP1:91,1] = PR[GP1:90,1] + -38.823;
   1:  PR[GP1:91,2] = PR[GP1:90,2] + -10.129;
   1:L PR[91] R[100]mm/sec CNT100;
   1:  PR[GP1:91,1] = PR[GP1:90,1] + -36.196;
   1:  PR[GP1:91,2] = PR[GP1:90,2] + -13.567;
   1:L PR[91] R[100]mm/sec CNT100;
   1:  PR[GP1:91,1] = PR[GP1:90,1] + -35.584;
   1:  PR[GP1:91,2] = PR[GP1:90,2] + -14.066;
   1:L PR[91] R[100]mm/sec CNT100;
   1:  PR[GP1:91,1] = PR[GP1:90,1] + -32.345;
   1:  PR[GP1:91,2] = PR[GP1:90,2] + -16.569;
   1:L PR[91] R[100]mm/sec CNT100;
   1:  PR[GP1:91,1] = PR[GP1:90,1] + -31.336;
   1:  PR[GP1:91,2] = PR[GP1:90,2] + -17.036;
   1:L PR[91] R[100]mm/sec CNT100;
   1:  PR[GP1:91,1] = PR[GP1:90,1] + -27.871;
   1:  PR[GP1:91,2] = PR[GP1:90,2] + -18.501;
   1:L PR[91] R[100]mm/sec CNT100;
   1:  PR[GP1:91,1] = PR[GP1:90,1] + -26.375;
   1:  PR[GP1:91,2] = PR[GP1:90,2] + -18.779;
   1:L PR[91] R[100]mm/sec CNT100;
   1:  PR[GP1:91,1] = PR[GP1:90,1] + -23.076;
   1:  PR[GP1:91,2] = PR[GP1:90,2] + -19.252;
   1:L PR[91] R[100]mm/sec CNT100;
   1:  PR[GP1:91,1] = PR[GP1:90,1] + -21.073;
   1:  PR[GP1:91,2] = PR[GP1:90,2] + -19.121;
   1:L PR[91] R[100]mm/sec CNT100;
   1:  PR[GP1:91,1] = PR[GP1:90,1] + -18.273;
   1:  PR[GP1:91,2] = PR[GP1:90,2] + -18.798;
   1:L PR[91] R[100]mm/sec CNT100;
   1:  PR[GP1:91,1] = PR[GP1:90,1] + -15.857;
   1:  PR[GP1:91,2] = PR[GP1:90,2] + -18.012;
   1:L PR[91] R[100]mm/sec CNT100;
   1:  PR[GP1:91,1] = PR[GP1:90,1] + -13.761;
